LIN {X 0,Y 509.786,Z 447.475,A -85,B 0,C 180,E1 -5449.613,E2 -5449.613} C_VEL
LIN {X 0,Y 509.778,Z 447.48,A -85,B 0,C 180,E1 -5452.656,E2 -5452.656} C_VEL
LIN {X 0,Y 509.83,Z 447.482,A -85,B 0,C 180,E1 -5455.803,E2 -5455.803} C_VEL
LIN {X 0,Y 509.837,Z 447.476,A -85,B 0,C 180,E1 -5458.723,E2 -5458.723} C_VEL
LIN {X 0,Y 509.815,Z 447.48,A -85,B 0,C 180,E1 -5461.152,E2 -5461.152} C_VEL
LIN {X 0,Y 509.86,Z 447.686,A -85,B 0,C 180,E1 -5463.635,E2 -5463.635} C_VEL
LIN {X 0,Y 511.214,Z 455.666,A -85,B 0,C 180,E1 -5465.408,E2 -5465.408} C_VEL
LIN {X 0,Y 510.839,Z 468.185,A -85,B 0,C 180,E1 -5467.982,E2 -5467.982} C_VEL
LIN {X 0,Y 510.48,Z 482.835,A -85,B 0,C 180,E1 -5470.915,E2 -5470.915} C_VEL
LIN {X 0,Y 510.057,Z 498.364,A -85,B 0,C 180,E1 -5474.004,E2 -5474.004} C_VEL
LIN {X 0,Y 510.013,Z 500.382,A -85,B 0,C 180,E1 -5474.39,E2 -5474.39} C_VEL
LIN {X 0,Y 510.872,Z 505.663,A -85,B 0,C 180,E1 -5474.531,E2 -5474.531} C_VEL
LIN {X 0,Y 512.207,Z 513.365,A -85,B 0,C 180,E1 -5474.681,E2 -5474.681} C_VEL
LIN {X 0,Y 511.746,Z 605.354,A -85,B 0,C 180,E1 -5475.993,E2 -5475.993} C_VEL
LIN {X 0,Y 511.617,Z 615.274,A -85,B 0,C 180,E1 -5476.217,E2 -5476.217} C_VEL
LIN {X 0,Y 511.372,Z 625.264,A -85,B 0,C 180,E1 -5476.539,E2 -5476.539} C_VEL
LIN {X 0,Y 511.129,Z 635.625,A -85,B 0,C 180,E1 -5476.988,E2 -5476.988} C_VEL
LIN {X 0,Y 510.913,Z 644.923,A -85,B 0,C 180,E1 -5477.497,E2 -5477.497} C_VEL
LIN {X 0,Y 510.669,Z 653.783,A -85,B 0,C 180,E1 -5478.087,E2 -5478.087} C_VEL
LIN {X 0,Y 510.376,Z 662.514,A -85,B 0,C 180,E1 -5478.784,E2 -5478.784} C_VEL
LIN {X 0,Y 510.112,Z 669.938,A -85,B 0,C 180,E1 -5479.482,E2 -5479.482} C_VEL
LIN {X 0,Y 509.84,Z 678.737,A -85,B 0,C 180,E1 -5480.479,E2 -5480.479} C_VEL
LIN {X 0,Y 509.675,Z 684.729,A -85,B 0,C 180,E1 -5481.276,E2 -5481.276} C_VEL
LIN {X 0,Y 509.495,Z 691.04,A -85,B 0,C 180,E1 -5482.271,E2 -5482.271} C_VEL
LIN {X 0,Y 509.351,Z 697.115,A -85,B 0,C 180,E1 -5483.443,E2 -5483.443} C_VEL
LIN {X 0,Y 509.296,Z 701.404,A -85,B 0,C 180,E1 -5484.457,E2 -5484.457} C_VEL
LIN {X 0,Y 509.206,Z 705.362,A -85,B 0,C 180,E1 -5485.647,E2 -5485.647} C_VEL
LIN {X 0,Y 509.201,Z 708.291,A -85,B 0,C 180,E1 -5486.835,E2 -5486.835} C_VEL
LIN {X 0,Y 509.19,Z 709.788,A -85,B 0,C 180,E1 -5487.627,E2 -5487.627} C_VEL
LIN {X 0,Y 509.074,Z 711.303,A -85,B 0,C 180,E1 -5489.209,E2 -5489.209} C_VEL
LIN {X 0,Y 509.066,Z 711.581,A -85,B 0,C 180,E1 -5490,E2 -5490} C_VEL
LIN {X 0,Y 509.113,Z 710.71,A -85,B 0,C 180,E1 -5491.582,E2 -5491.582} C_VEL
LIN {X 0,Y 509.19,Z 709.788,A -85,B 0,C 180,E1 -5492.373,E2 -5492.373} C_VEL
LIN {X 0,Y 509.246,Z 706.45,A -85,B 0,C 180,E1 -5493.957,E2 -5493.957} C_VEL
LIN {X 0,Y 509.244,Z 702.829,A -85,B 0,C 180,E1 -5495.147,E2 -5495.147} C_VEL
LIN {X 0,Y 509.343,Z 699.891,A -85,B 0,C 180,E1 -5495.94,E2 -5495.94} C_VEL
LIN {X 0,Y 509.421,Z 694.317,A -85,B 0,C 180,E1 -5497.132,E2 -5497.132} C_VEL
LIN {X 0,Y 509.573,Z 688.665,A -85,B 0,C 180,E1 -5498.127,E2 -5498.127} C_VEL
LIN {X 0,Y 509.755,Z 681.86,A -85,B 0,C 180,E1 -5499.123,E2 -5499.123} C_VEL
LIN {X 0,Y 509.978,Z 673.64,A -85,B 0,C 180,E1 -5500.12,E2 -5500.12} C_VEL
LIN {X 0,Y 510.273,Z 665.811,A -85,B 0,C 180,E1 -5500.916,E2 -5500.916} C_VEL
LIN {X 0,Y 510.584,Z 657.725,A -85,B 0,C 180,E1 -5501.613,E2 -5501.613} C_VEL
LIN {X 0,Y 510.791,Z 647.557,A -85,B 0,C 180,E1 -5502.339,E2 -5502.339} C_VEL
LIN {X 0,Y 511.061,Z 639.564,A -85,B 0,C 180,E1 -5502.812,E2 -5502.812} C_VEL
LIN {X 0,Y 511.326,Z 629.054,A -85,B 0,C 180,E1 -5503.31,E2 -5503.31} C_VEL
LIN {X 0,Y 511.559,Z 618.719,A -85,B 0,C 180,E1 -5503.683,E2 -5503.683} C_VEL
LIN {X 0,Y 511.694,Z 607.997,A -85,B 0,C 180,E1 -5503.958,E2 -5503.958} C_VEL
LIN {X 0,Y 511.904,Z 585.223,A -85,B 0,C 180,E1 -5504.307,E2 -5504.307} C_VEL
LIN {X 0,Y 512.124,Z 512.714,A -85,B 0,C 180,E1 -5505.33,E2 -5505.33} C_VEL
LIN {X 0,Y 510.034,Z 500.586,A -85,B 0,C 180,E1 -5505.592,E2 -5505.592} C_VEL
LIN {X 0,Y 510.478,Z 483.881,A -85,B 0,C 180,E1 -5508.877,E2 -5508.877} C_VEL
LIN {X 0,Y 510.831,Z 469.232,A -85,B 0,C 180,E1 -5511.806,E2 -5511.806} C_VEL
LIN {X 0,Y 511.246,Z 456.791,A -85,B 0,C 180,E1 -5514.356,E2 -5514.356} C_VEL
LIN {X 0,Y 510.607,Z 451.626,A -85,B 0,C 180,E1 -5515.475,E2 -5515.475} C_VEL
LIN {X 0,Y 509.819,Z 447.591,A -85,B 0,C 180,E1 -5516.421,E2 -5516.421} C_VEL
LIN {X 0,Y 509.815,Z 447.48,A -85,B 0,C 180,E1 -5518.848,E2 -5518.848} C_VEL
LIN {X 0,Y 509.811,Z 447.481,A -85,B 0,C 180,E1 -5521.59,E2 -5521.59} C_VEL
LIN {X 0,Y 509.834,Z 447.478,A -85,B 0,C 180,E1 -5524.414,E2 -5524.414} C_VEL
LIN {X 0,Y 509.778,Z 447.48,A -85,B 0,C 180,E1 -5527.344,E2 -5527.344} C_VEL
LIN {X 0,Y 509.786,Z 447.475,A -85,B 0,C 180,E1 -5530.387,E2 -5530.387} C_VEL
LIN {X 0,Y 509.792,Z 447.48,A -85,B 0,C 180,E1 -5533.574,E2 -5533.574} C_VEL
LIN {X 0,Y 509.791,Z 447.483,A -85,B 0,C 180,E1 -5536.424,E2 -5536.424} C_VEL
LIN {X 0,Y 509.785,Z 447.481,A -85,B 0,C 180,E1 -5539.612,E2 -5539.612} C_VEL
LIN {X 0,Y 509.775,Z 447.482,A -85,B 0,C 180,E1 -5542.655,E2 -5542.655} C_VEL
LIN {X 0,Y 509.837,Z 447.474,A -85,B 0,C 180,E1 -5545.8,E2 -5545.8} C_VEL
LIN {X 0,Y 509.835,Z 447.474,A -85,B 0,C 180,E1 -5548.721,E2 -5548.721} C_VEL
LIN {X 0,Y 509.831,Z 447.472,A -85,B 0,C 180,E1 -5551.152,E2 -5551.152} C_VEL
LIN {X 0,Y 509.834,Z 447.469,A -85,B 0,C 180,E1 -5553.824,E2 -5553.824} C_VEL
LIN {X 0,Y 509.815,Z 447.479,A -85,B 0,C 180,E1 -5556.435,E2 -5556.435} C_VEL
LIN {X 0,Y 509.817,Z 447.475,A -85,B 0,C 180,E1 -5559.618,E2 -5559.618} C_VEL
LIN {X 0,Y 509.845,Z 447.471,A -85,B 0,C 180,E1 -5562.345,E2 -5562.345} C_VEL
LIN {X 0,Y 509.817,Z 447.477,A -85,B 0,C 180,E1 -5565.632,E2 -5565.632} C_VEL
LIN {X 0,Y 509.886,Z 447.469,A -85,B 0,C 180,E1 -5568.13,E2 -5568.13} C_VEL
LIN {X 0,Y 509.867,Z 447.458,A -85,B 0,C 180,E1 -5571.278,E2 -5571.278} C_VEL
LIN {X 0,Y 509.91,Z 447.463,A -85,B 0,C 180,E1 -5573.668,E2 -5573.668} C_VEL
LIN {X 0,Y 509.876,Z 447.467,A -85,B 0,C 180,E1 -5576.838,E2 -5576.838} C_VEL
LIN {X 0,Y 509.916,Z 447.46,A -85,B 0,C 180,E1 -5578.419,E2 -5578.419} C_VEL
LIN {X 0,Y 510.027,Z 447.445,A -85,B 0,C 180,E1 -5579.999,E2 -5579.999} C_VEL
LIN {X 0,Y 510.034,Z 447.45,A -85,B 0,C 180,E1 -5582.368,E2 -5582.368} C_VEL
LIN {X 0,Y 509.929,Z 447.463,A -85,B 0,C 180,E1 -5585.535,E2 -5585.535} C_VEL
LIN {X 0,Y 509.867,Z 447.474,A -85,B 0,C 180,E1 -5587.922,E2 -5587.922} C_VEL
LIN {X 0,Y 509.852,Z 447.463,A -85,B 0,C 180,E1 -5591.125,E2 -5591.125} C_VEL
LIN {X 0,Y 509.818,Z 447.475,A -85,B 0,C 180,E1 -5593.552,E2 -5593.552} C_VEL
LIN {X 0,Y 509.787,Z 447.487,A -85,B 0,C 180,E1 -5596.004,E2 -5596.004} C_VEL
LIN {X 0,Y 509.805,Z 447.469,A -85,B 0,C 180,E1 -5598.484,E2 -5598.484} C_VEL
LIN {X 0,Y 509.822,Z 447.471,A -85,B 0,C 180,E1 -5601.001,E2 -5601.001} C_VEL
LIN {X 0,Y 509.807,Z 447.479,A -85,B 0,C 180,E1 -5603.563,E2 -5603.563} C_VEL
LIN {X 0,Y 509.795,Z 447.475,A -85,B 0,C 180,E1 -5606.353,E2 -5606.353} C_VEL
LIN {X 0,Y 509.821,Z 447.472,A -85,B 0,C 180,E1 -5608.846,E2 -5608.846} C_VEL
LIN {X 0,Y 509.79,Z 447.482,A -85,B 0,C 180,E1 -5611.59,E2 -5611.59} C_VEL
LIN {X 0,Y 509.82,Z 447.473,A -85,B 0,C 180,E1 -5614.414,E2 -5614.414} C_VEL
LIN {X 0,Y 509.766,Z 447.483,A -85,B 0,C 180,E1 -5617.343,E2 -5617.343} C_VEL
LIN {X 0,Y 509.799,Z 447.477,A -85,B 0,C 180,E1 -5620.384,E2 -5620.384} C_VEL
LIN {X 0,Y 509.79,Z 447.481,A -85,B 0,C 180,E1 -5623.573,E2 -5623.573} C_VEL
LIN {X 0,Y 509.777,Z 447.473,A -85,B 0,C 180,E1 -5626.424,E2 -5626.424} C_VEL
LIN {X 0,Y 509.77,Z 447.475,A -85,B 0,C 180,E1 -5629.612,E2 -5629.612} C_VEL
LIN {X 0,Y 509.763,Z 447.483,A -85,B 0,C 180,E1 -5632.655,E2 -5632.655} C_VEL
LIN {X 0,Y 509.749,Z 447.486,A -85,B 0,C 180,E1 -5633.7,E2 -5633.7} C_VEL
LIN {X 0,Y 509.095,Z 447.56,A -85,B 0,C 180,E1 -5634.361,E2 -5634.361} C_VEL
LIN {X 0,Y 506.291,Z 447.907,A -85,B 0,C 180,E1 -5635.433,E2 -5635.433} C_VEL
LIN {X 0,Y 503.905,Z 448.213,A -85,B 0,C 180,E1 -5636.297,E2 -5636.297} C_VEL
LIN {X 0,Y 502.86,Z 448.341,A -85,B 0,C 180,E1 -5636.964,E2 -5636.964} C_VEL
LIN {X 0,Y 502.764,Z 448.353,A -85,B 0,C 180,E1 -5637.189,E2 -5637.189} C_VEL
LIN {X 0,Y 502.793,Z 448.35,A -85,B 0,C 180,E1 -5640.066,E2 -5640.066} C_VEL
LIN {X 0,Y 502.757,Z 448.358,A -85,B 0,C 180,E1 -5643.459,E2 -5643.459} C_VEL
LIN {X 0,Y 502.749,Z 448.364,A -85,B 0,C 180,E1 -5646.084,E2 -5646.084} C_VEL
LIN {X 0,Y 502.761,Z 448.357,A -85,B 0,C 180,E1 -5648.688,E2 -5648.688} C_VEL
LIN {X 0,Y 502.79,Z 448.353,A -85,B 0,C 180,E1 -5651.247,E2 -5651.247} C_VEL
LIN {X 0,Y 502.818,Z 448.35,A -85,B 0,C 180,E1 -5654.664,E2 -5654.664} C_VEL
LIN {X 0,Y 502.852,Z 448.351,A -85,B 0,C 180,E1 -5658.043,E2 -5658.043} C_VEL
LIN {X 0,Y 502.829,Z 448.349,A -85,B 0,C 180,E1 -5661.156,E2 -5661.156} C_VEL
LIN {X 0,Y 502.853,Z 448.349,A -85,B 0,C 180,E1 -5663.58,E2 -5663.58} C_VEL
LIN {X 0,Y 502.814,Z 448.351,A -85,B 0,C 180,E1 -5666.795,E2 -5666.795} C_VEL
LIN {X 0,Y 502.875,Z 448.346,A -85,B 0,C 180,E1 -5668.398,E2 -5668.398} C_VEL
LIN {X 0,Y 502.986,Z 448.335,A -85,B 0,C 180,E1 -5670,E2 -5670} C_VEL
LIN {X 0,Y 502.992,Z 448.331,A -85,B 0,C 180,E1 -5672.402,E2 -5672.402} C_VEL
LIN {X 0,Y 502.877,Z 448.346,A -85,B 0,C 180,E1 -5675.614,E2 -5675.614} C_VEL
LIN {X 0,Y 502.831,Z 448.354,A -85,B 0,C 180,E1 -5678.034,E2 -5678.034} C_VEL
LIN {X 0,Y 502.82,Z 448.35,A -85,B 0,C 180,E1 -5681.284,E2 -5681.284} C_VEL
LIN {X 0,Y 502.812,Z 448.352,A -85,B 0,C 180,E1 -5684.572,E2 -5684.572} C_VEL
LIN {X 0,Y 502.792,Z 448.359,A -85,B 0,C 180,E1 -5688.109,E2 -5688.109} C_VEL
LIN {X 0,Y 502.813,Z 448.351,A -85,B 0,C 180,E1 -5690.537,E2 -5690.537} C_VEL
LIN {X 0,Y 502.769,Z 448.355,A -85,B 0,C 180,E1 -5693.041,E2 -5693.041} C_VEL
LIN {X 0,Y 502.758,Z 448.361,A -85,B 0,C 180,E1 -5695.68,E2 -5695.68} C_VEL
LIN {X 0,Y 502.753,Z 448.353,A -85,B 0,C 180,E1 -5698.378,E2 -5698.378} C_VEL
LIN {X 0,Y 502.768,Z 448.354,A -85,B 0,C 180,E1 -5701.145,E2 -5701.145} C_VEL
LIN {X 0,Y 502.767,Z 448.35,A -85,B 0,C 180,E1 -5703.996,E2 -5703.996} C_VEL
LIN {X 0,Y 502.716,Z 448.36,A -85,B 0,C 180,E1 -5707.171,E2 -5707.171} C_VEL
LIN {X 0,Y 502.717,Z 448.358,A -85,B 0,C 180,E1 -5710.021,E2 -5710.021} C_VEL
LIN {X 0,Y 502.724,Z 448.348,A -85,B 0,C 180,E1 -5713.236,E2 -5713.236} C_VEL
LIN {X 0,Y 502.764,Z 448.356,A -85,B 0,C 180,E1 -5715.661,E2 -5715.661} C_VEL
LIN {X 0,Y 502.75,Z 448.351,A -85,B 0,C 180,E1 -5719.013,E2 -5719.013} C_VEL
LIN {X 0,Y 502.746,Z 448.364,A -85,B 0,C 180,E1 -5722.044,E2 -5722.044} C_VEL
LIN {X 0,Y 502.769,Z 448.348,A -85,B 0,C 180,E1 -5725.034,E2 -5725.034} C_VEL
LIN {X 0,Y 502.751,Z 448.362,A -85,B 0,C 180,E1 -5727.915,E2 -5727.915} C_VEL
LIN {X 0,Y 502.79,Z 448.348,A -85,B 0,C 180,E1 -5730.712,E2 -5730.712} C_VEL
LIN {X 0,Y 502.76,Z 448.349,A -85,B 0,C 180,E1 -5733.462,E2 -5733.462} C_VEL
LIN {X 0,Y 502.755,Z 448.362,A -85,B 0,C 180,E1 -5736.086,E2 -5736.086} C_VEL
LIN {X 0,Y 502.761,Z 448.351,A -85,B 0,C 180,E1 -5738.689,E2 -5738.689} C_VEL
LIN {X 0,Y 502.777,Z 448.35,A -85,B 0,C 180,E1 -5741.9,E2 -5741.9} C_VEL
LIN {X 0,Y 502.817,Z 448.349,A -85,B 0,C 180,E1 -5745.43,E2 -5745.43} C_VEL
LIN {X 0,Y 502.828,Z 448.337,A -85,B 0,C 180,E1 -5748.717,E2 -5748.717} C_VEL
LIN {X 0,Y 502.838,Z 448.346,A -85,B 0,C 180,E1 -5751.967,E2 -5751.967} C_VEL
LIN {X 0,Y 502.886,Z 448.341,A -85,B 0,C 180,E1 -5754.387,E2 -5754.387} C_VEL
LIN {X 0,Y 503.001,Z 448.325,A -85,B 0,C 180,E1 -5757.599,E2 -5757.599} C_VEL
LIN {X 0,Y 502.996,Z 448.32,A -85,B 0,C 180,E1 -5760.001,E2 -5760.001} C_VEL
LIN {X 0,Y 503.002,Z 448.325,A -85,B 0,C 180,E1 -5762.404,E2 -5762.404} C_VEL
LIN {X 0,Y 502.886,Z 448.343,A -85,B 0,C 180,E1 -5765.615,E2 -5765.615} C_VEL
LIN {X 0,Y 502.841,Z 448.34,A -85,B 0,C 180,E1 -5768.035,E2 -5768.035} C_VEL
LIN {X 0,Y 502.832,Z 448.34,A -85,B 0,C 180,E1 -5771.285,E2 -5771.285} C_VEL
LIN {X 0,Y 502.795,Z 448.349,A -85,B 0,C 180,E1 -5774.573,E2 -5774.573} C_VEL
LIN {X 0,Y 502.784,Z 448.346,A -85,B 0,C 180,E1 -5778.102,E2 -5778.102} C_VEL
LIN {X 0,Y 502.757,Z 448.353,A -85,B 0,C 180,E1 -5781.313,E2 -5781.313} C_VEL
LIN {X 0,Y 502.763,Z 448.359,A -85,B 0,C 180,E1 -5783.916,E2 -5783.916} C_VEL
LIN {X 0,Y 502.779,Z 448.344,A -85,B 0,C 180,E1 -5786.572,E2 -5786.572} C_VEL
LIN {X 0,Y 502.808,Z 448.357,A -85,B 0,C 180,E1 -5789.935,E2 -5789.935} C_VEL
LIN {X 0,Y 502.797,Z 448.346,A -85,B 0,C 180,E1 -5793.035,E2 -5793.035} C_VEL
LIN {X 0,Y 502.743,Z 448.363,A -85,B 0,C 180,E1 -5795.955,E2 -5795.955} C_VEL
LIN {X 0,Y 502.767,Z 448.351,A -85,B 0,C 180,E1 -5798.98,E2 -5798.98} C_VEL
LIN {X 0,Y 502.745,Z 448.361,A -85,B 0,C 180,E1 -5802.193,E2 -5802.193} C_VEL
LIN {X 0,Y 502.778,Z 448.355,A -85,B 0,C 180,E1 -5805.472,E2 -5805.472} C_VEL
LIN {X 0,Y 502.75,Z 448.347,A -85,B 0,C 180,E1 -5808.928,E2 -5808.928} C_VEL
LIN {X 0,Y 502.759,Z 448.36,A -85,B 0,C 180,E1 -5812.043,E2 -5812.043} C_VEL
LIN {X 0,Y 502.753,Z 448.355,A -85,B 0,C 180,E1 -5815.031,E2 -5815.031} C_VEL
LIN {X 0,Y 502.762,Z 448.36,A -85,B 0,C 180,E1 -5817.914,E2 -5817.914} C_VEL
LIN {X 0,Y 502.782,Z 448.356,A -85,B 0,C 180,E1 -5820.71,E2 -5820.71} C_VEL
LIN {X 0,Y 502.819,Z 448.562,A -85,B 0,C 180,E1 -5823.451,E2 -5823.451} C_VEL
LIN {X 0,Y 504.244,Z 456.649,A -85,B 0,C 180,E1 -5825.284,E2 -5825.284} C_VEL
LIN {X 0,Y 503.906,Z 468.046,A -85,B 0,C 180,E1 -5827.663,E2 -5827.663} C_VEL
LIN {X 0,Y 503.51,Z 481.652,A -85,B 0,C 180,E1 -5830.428,E2 -5830.428} C_VEL
LIN {X 0,Y 503.131,Z 495.1,A -85,B 0,C 180,E1 -5833.151,E2 -5833.151} C_VEL
LIN {X 0,Y 503.005,Z 500.389,A -85,B 0,C 180,E1 -5834.185,E2 -5834.185} C_VEL
LIN {X 0,Y 505.356,Z 514.508,A -85,B 0,C 180,E1 -5834.488,E2 -5834.488} C_VEL
LIN {X 0,Y 504.87,Z 605.158,A -85,B 0,C 180,E1 -5835.798,E2 -5835.798} C_VEL
LIN {X 0,Y 504.721,Z 615.078,A -85,B 0,C 180,E1 -5836.025,E2 -5836.025} C_VEL
LIN {X 0,Y 504.459,Z 625.067,A -85,B 0,C 180,E1 -5836.351,E2 -5836.351} C_VEL
LIN {X 0,Y 504.181,Z 635.428,A -85,B 0,C 180,E1 -5836.806,E2 -5836.806} C_VEL
LIN {X 0,Y 503.952,Z 645.118,A -85,B 0,C 180,E1 -5837.347,E2 -5837.347} C_VEL
LIN {X 0,Y 503.676,Z 653.586,A -85,B 0,C 180,E1 -5837.919,E2 -5837.919} C_VEL
LIN {X 0,Y 503.397,Z 662.317,A -85,B 0,C 180,E1 -5838.627,E2 -5838.627} C_VEL
LIN {X 0,Y 503.107,Z 669.741,A -85,B 0,C 180,E1 -5839.334,E2 -5839.334} C_VEL
LIN {X 0,Y 502.808,Z 678.54,A -85,B 0,C 180,E1 -5840.344,E2 -5840.344} C_VEL
LIN {X 0,Y 502.61,Z 684.531,A -85,B 0,C 180,E1 -5841.152,E2 -5841.152} C_VEL
LIN {X 0,Y 502.421,Z 690.843,A -85,B 0,C 180,E1 -5842.161,E2 -5842.161} C_VEL
LIN {X 0,Y 502.318,Z 696.295,A -85,B 0,C 180,E1 -5843.21,E2 -5843.21} C_VEL
LIN {X 0,Y 502.214,Z 701.207,A -85,B 0,C 180,E1 -5844.378,E2 -5844.378} C_VEL
LIN {X 0,Y 502.104,Z 705.165,A -85,B 0,C 180,E1 -5845.585,E2 -5845.585} C_VEL
LIN {X 0,Y 502.121,Z 708.095,A -85,B 0,C 180,E1 -5846.791,E2 -5846.791} C_VEL
LIN {X 0,Y 502.092,Z 709.591,A -85,B 0,C 180,E1 -5847.593,E2 -5847.593} C_VEL
LIN {X 0,Y 501.991,Z 711.107,A -85,B 0,C 180,E1 -5849.198,E2 -5849.198} C_VEL
LIN {X 0,Y 501.98,Z 711.385,A -85,B 0,C 180,E1 -5850,E2 -5850} C_VEL
LIN {X 0,Y 502.037,Z 710.515,A -85,B 0,C 180,E1 -5851.604,E2 -5851.604} C_VEL
LIN {X 0,Y 502.092,Z 709.591,A -85,B 0,C 180,E1 -5852.407,E2 -5852.407} C_VEL
LIN {X 0,Y 502.139,Z 706.253,A -85,B 0,C 180,E1 -5854.013,E2 -5854.013} C_VEL
LIN {X 0,Y 502.175,Z 702.633,A -85,B 0,C 180,E1 -5855.219,E2 -5855.219} C_VEL
LIN {X 0,Y 502.237,Z 697.904,A -85,B 0,C 180,E1 -5856.427,E2 -5856.427} C_VEL
LIN {X 0,Y 502.362,Z 693.027,A -85,B 0,C 180,E1 -5857.435,E2 -5857.435} C_VEL
LIN {X 0,Y 502.529,Z 687.155,A -85,B 0,C 180,E1 -5858.444,E2 -5858.444} C_VEL
LIN {X 0,Y 502.699,Z 681.662,A -85,B 0,C 180,E1 -5859.252,E2 -5859.252} C_VEL
LIN {X 0,Y 502.958,Z 673.443,A -85,B 0,C 180,E1 -5860.262,E2 -5860.262} C_VEL
LIN {X 0,Y 503.276,Z 665.614,A -85,B 0,C 180,E1 -5861.07,E2 -5861.07} C_VEL
LIN {X 0,Y 503.605,Z 657.528,A -85,B 0,C 180,E1 -5861.777,E2 -5861.777} C_VEL
LIN {X 0,Y 503.803,Z 648.403,A -85,B 0,C 180,E1 -5862.446,E2 -5862.446} C_VEL
LIN {X 0,Y 504.119,Z 639.367,A -85,B 0,C 180,E1 -5862.991,E2 -5862.991} C_VEL
LIN {X 0,Y 504.42,Z 628.858,A -85,B 0,C 180,E1 -5863.496,E2 -5863.496} C_VEL
LIN {X 0,Y 504.664,Z 618.523,A -85,B 0,C 180,E1 -5863.874,E2 -5863.874} C_VEL
LIN {X 0,Y 504.803,Z 607.8,A -85,B 0,C 180,E1 -5864.153,E2 -5864.153} C_VEL
LIN {X 0,Y 505.041,Z 585.027,A -85,B 0,C 180,E1 -5864.506,E2 -5864.506} C_VEL
LIN {X 0,Y 505.312,Z 513.673,A -85,B 0,C 180,E1 -5865.526,E2 -5865.526} C_VEL
LIN {X 0,Y 503.03,Z 500.529,A -85,B 0,C 180,E1 -5865.806,E2 -5865.806} C_VEL
LIN {X 0,Y 503.006,Z 499.492,A -85,B 0,C 180,E1 -5865.945,E2 -5865.945} C_VEL
LIN {X 0,Y 503.457,Z 484.79,A -85,B 0,C 180,E1 -5868.939,E2 -5868.939} C_VEL
LIN {X 0,Y 503.874,Z 469.094,A -85,B 0,C 180,E1 -5872.123,E2 -5872.123} C_VEL
LIN {X 0,Y 504.288,Z 457.707,A -85,B 0,C 180,E1 -5874.494,E2 -5874.494} C_VEL
LIN {X 0,Y 503.382,Z 451.532,A -85,B 0,C 180,E1 -5875.863,E2 -5875.863} C_VEL
LIN {X 0,Y 502.788,Z 448.45,A -85,B 0,C 180,E1 -5876.626,E2 -5876.626} C_VEL
LIN {X 0,Y 502.79,Z 448.356,A -85,B 0,C 180,E1 -5879.929,E2 -5879.929} C_VEL
LIN {X 0,Y 502.804,Z 448.348,A -85,B 0,C 180,E1 -5883.033,E2 -5883.033} C_VEL
LIN {X 0,Y 502.744,Z 448.358,A -85,B 0,C 180,E1 -5885.953,E2 -5885.953} C_VEL
LIN {X 0,Y 502.774,Z 448.353,A -85,B 0,C 180,E1 -5888.978,E2 -5888.978} C_VEL
LIN {X 0,Y 502.745,Z 448.359,A -85,B 0,C 180,E1 -5892.191,E2 -5892.191} C_VEL
LIN {X 0,Y 502.778,Z 448.352,A -85,B 0,C 180,E1 -5895.47,E2 -5895.47} C_VEL
LIN {X 0,Y 502.749,Z 448.355,A -85,B 0,C 180,E1 -5898.926,E2 -5898.926} C_VEL
LIN {X 0,Y 502.754,Z 448.361,A -85,B 0,C 180,E1 -5902.042,E2 -5902.042} C_VEL
LIN {X 0,Y 502.781,Z 448.348,A -85,B 0,C 180,E1 -5905.032,E2 -5905.032} C_VEL
LIN {X 0,Y 502.762,Z 448.356,A -85,B 0,C 180,E1 -5907.913,E2 -5907.913} C_VEL
LIN {X 0,Y 502.801,Z 448.349,A -85,B 0,C 180,E1 -5910.71,E2 -5910.71} C_VEL
LIN {X 0,Y 502.77,Z 448.345,A -85,B 0,C 180,E1 -5913.459,E2 -5913.459} C_VEL
LIN {X 0,Y 502.763,Z 448.359,A -85,B 0,C 180,E1 -5916.084,E2 -5916.084} C_VEL
LIN {X 0,Y 502.757,Z 448.353,A -85,B 0,C 180,E1 -5918.687,E2 -5918.687} C_VEL
LIN {X 0,Y 502.784,Z 448.346,A -85,B 0,C 180,E1 -5921.898,E2 -5921.898} C_VEL
LIN {X 0,Y 502.795,Z 448.349,A -85,B 0,C 180,E1 -5925.427,E2 -5925.427} C_VEL
LIN {X 0,Y 502.832,Z 448.34,A -85,B 0,C 180,E1 -5928.715,E2 -5928.715} C_VEL
LIN {X 0,Y 502.841,Z 448.34,A -85,B 0,C 180,E1 -5931.965,E2 -5931.965} C_VEL
LIN {X 0,Y 502.886,Z 448.343,A -85,B 0,C 180,E1 -5934.385,E2 -5934.385} C_VEL
LIN {X 0,Y 503.002,Z 448.325,A -85,B 0,C 180,E1 -5937.596,E2 -5937.596} C_VEL
LIN {X 0,Y 502.996,Z 448.32,A -85,B 0,C 180,E1 -5939.999,E2 -5939.999} C_VEL
LIN {X 0,Y 503.001,Z 448.325,A -85,B 0,C 180,E1 -5942.401,E2 -5942.401} C_VEL
LIN {X 0,Y 502.886,Z 448.341,A -85,B 0,C 180,E1 -5945.613,E2 -5945.613} C_VEL
LIN {X 0,Y 502.838,Z 448.346,A -85,B 0,C 180,E1 -5948.033,E2 -5948.033} C_VEL
LIN {X 0,Y 502.828,Z 448.337,A -85,B 0,C 180,E1 -5951.283,E2 -5951.283} C_VEL
LIN {X 0,Y 502.817,Z 448.349,A -85,B 0,C 180,E1 -5954.57,E2 -5954.57} C_VEL
LIN {X 0,Y 502.777,Z 448.35,A -85,B 0,C 180,E1 -5958.1,E2 -5958.1} C_VEL
LIN {X 0,Y 502.761,Z 448.351,A -85,B 0,C 180,E1 -5961.311,E2 -5961.311} C_VEL
LIN {X 0,Y 502.755,Z 448.362,A -85,B 0,C 180,E1 -5963.914,E2 -5963.914} C_VEL
LIN {X 0,Y 502.77,Z 448.347,A -85,B 0,C 180,E1 -5966.57,E2 -5966.57} C_VEL
LIN {X 0,Y 502.797,Z 448.354,A -85,B 0,C 180,E1 -5969.933,E2 -5969.933} C_VEL
LIN {X 0,Y 502.786,Z 448.349,A -85,B 0,C 180,E1 -5973.033,E2 -5973.033} C_VEL
LIN {X 0,Y 502.731,Z 448.36,A -85,B 0,C 180,E1 -5975.953,E2 -5975.953} C_VEL
LIN {X 0,Y 502.769,Z 448.353,A -85,B 0,C 180,E1 -5978.977,E2 -5978.977} C_VEL
LIN {X 0,Y 502.73,Z 448.365,A -85,B 0,C 180,E1 -5982.191,E2 -5982.191} C_VEL
LIN {X 0,Y 502.763,Z 448.354,A -85,B 0,C 180,E1 -5985.47,E2 -5985.47} C_VEL
LIN {X 0,Y 502.734,Z 448.348,A -85,B 0,C 180,E1 -5988.926,E2 -5988.926} C_VEL
LIN {X 0,Y 502.743,Z 448.366,A -85,B 0,C 180,E1 -5992.042,E2 -5992.042} C_VEL
LIN {X 0,Y 502.766,Z 448.344,A -85,B 0,C 180,E1 -5995.032,E2 -5995.032} C_VEL
LIN {X 0,Y 502.764,Z 448.353,A -85,B 0,C 180,E1 -5997.189,E2 -5997.189} C_VEL
LIN {X 0,Y 502.071,Z 448.447,A -85,B 0,C 180,E1 -5997.858,E2 -5997.858} C_VEL
LIN {X 0,Y 499.221,Z 448.795,A -85,B 0,C 180,E1 -5998.944,E2 -5998.944} C_VEL
LIN {X 0,Y 496.826,Z 449.096,A -85,B 0,C 180,E1 -5999.82,E2 -5999.82} C_VEL
LIN {X 0,Y 495.794,Z 449.218,A -85,B 0,C 180,E1 -6000.495,E2 -6000.495} C_VEL
LIN {X 0,Y 495.707,Z 449.227,A -85,B 0,C 180,E1 -6000.724,E2 -6000.724} C_VEL
LIN {X 0,Y 495.699,Z 449.242,A -85,B 0,C 180,E1 -6003.927,E2 -6003.927} C_VEL
LIN {X 0,Y 495.741,Z 449.231,A -85,B 0,C 180,E1 -6007.14,E2 -6007.14} C_VEL
LIN {X 0,Y 495.743,Z 449.237,A -85,B 0,C 180,E1 -6010.109,E2 -6010.109} C_VEL
LIN {X 0,Y 495.692,Z 449.239,A -85,B 0,C 180,E1 -6012.678,E2 -6012.678} C_VEL
LIN {X 0,Y 495.762,Z 449.229,A -85,B 0,C 180,E1 -6015.216,E2 -6015.216} C_VEL
LIN {X 0,Y 495.804,Z 449.226,A -85,B 0,C 180,E1 -6018.554,E2 -6018.554} C_VEL
LIN {X 0,Y 495.795,Z 449.23,A -85,B 0,C 180,E1 -6021.851,E2 -6021.851} C_VEL
LIN {X 0,Y 495.836,Z 449.224,A -85,B 0,C 180,E1 -6024.306,E2 -6024.306} C_VEL
LIN {X 0,Y 495.959,Z 449.207,A -85,B 0,C 180,E1 -6027.564,E2 -6027.564} C_VEL
LIN {X 0,Y 495.955,Z 449.211,A -85,B 0,C 180,E1 -6030,E2 -6030} C_VEL
LIN {X 0,Y 495.959,Z 449.207,A -85,B 0,C 180,E1 -6032.436,E2 -6032.436} C_VEL
LIN {X 0,Y 495.836,Z 449.224,A -85,B 0,C 180,E1 -6035.694,E2 -6035.694} C_VEL
LIN {X 0,Y 495.795,Z 449.23,A -85,B 0,C 180,E1 -6038.149,E2 -6038.149} C_VEL
LIN {X 0,Y 495.804,Z 449.226,A -85,B 0,C 180,E1 -6041.446,E2 -6041.446} C_VEL
LIN {X 0,Y 495.762,Z 449.229,A -85,B 0,C 180,E1 -6044.784,E2 -6044.784} C_VEL
LIN {X 0,Y 495.755,Z 449.234,A -85,B 0,C 180,E1 -6048.235,E2 -6048.235} C_VEL
LIN {X 0,Y 495.758,Z 449.229,A -85,B 0,C 180,E1 -6050.757,E2 -6050.757} C_VEL
LIN {X 0,Y 495.721,Z 449.234,A -85,B 0,C 180,E1 -6053.388,E2 -6053.388} C_VEL
LIN {X 0,Y 495.721,Z 449.233,A -85,B 0,C 180,E1 -6056.73,E2 -6056.73} C_VEL
LIN {X 0,Y 495.739,Z 449.226,A -85,B 0,C 180,E1 -6059.748,E2 -6059.748} C_VEL
LIN {X 0,Y 495.726,Z 449.231,A -85,B 0,C 180,E1 -6062.597,E2 -6062.597} C_VEL
LIN {X 0,Y 495.712,Z 449.225,A -85,B 0,C 180,E1 -6065.54,E2 -6065.54} C_VEL
LIN {X 0,Y 495.718,Z 449.232,A -85,B 0,C 180,E1 -6068.765,E2 -6068.765} C_VEL
LIN {X 0,Y 495.686,Z 449.224,A -85,B 0,C 180,E1 -6071.788,E2 -6071.788} C_VEL
LIN {X 0,Y 495.721,Z 449.229,A -85,B 0,C 180,E1 -6075.142,E2 -6075.142} C_VEL
LIN {X 0,Y 495.709,Z 449.233,A -85,B 0,C 180,E1 -6078.216,E2 -6078.216} C_VEL
LIN {X 0,Y 495.726,Z 449.231,A -85,B 0,C 180,E1 -6081.236,E2 -6081.236} C_VEL
LIN {X 0,Y 495.715,Z 449.228,A -85,B 0,C 180,E1 -6084.462,E2 -6084.462} C_VEL
LIN {X 0,Y 495.73,Z 449.23,A -85,B 0,C 180,E1 -6087.405,E2 -6087.405} C_VEL
LIN {X 0,Y 495.744,Z 449.23,A -85,B 0,C 180,E1 -6090.254,E2 -6090.254} C_VEL
LIN {X 0,Y 495.726,Z 449.223,A -85,B 0,C 180,E1 -6093.272,E2 -6093.272} C_VEL
LIN {X 0,Y 495.728,Z 449.231,A -85,B 0,C 180,E1 -6096.613,E2 -6096.613} C_VEL
LIN {X 0,Y 495.758,Z 449.224,A -85,B 0,C 180,E1 -6099.329,E2 -6099.329} C_VEL
LIN {X 0,Y 495.726,Z 449.226,A -85,B 0,C 180,E1 -6101.828,E2 -6101.828} C_VEL
LIN {X 0,Y 495.767,Z 449.226,A -85,B 0,C 180,E1 -6105.218,E2 -6105.218} C_VEL
LIN {X 0,Y 495.813,Z 449.212,A -85,B 0,C 180,E1 -6108.555,E2 -6108.555} C_VEL
LIN {X 0,Y 495.802,Z 449.22,A -85,B 0,C 180,E1 -6111.852,E2 -6111.852} C_VEL
LIN {X 0,Y 495.844,Z 449.219,A -85,B 0,C 180,E1 -6114.307,E2 -6114.307} C_VEL
LIN {X 0,Y 495.968,Z 449.201,A -85,B 0,C 180,E1 -6117.565,E2 -6117.565} C_VEL
LIN {X 0,Y 495.965,Z 449.195,A -85,B 0,C 180,E1 -6120.001,E2 -6120.001} C_VEL
LIN {X 0,Y 495.969,Z 449.201,A -85,B 0,C 180,E1 -6122.438,E2 -6122.438} C_VEL
LIN {X 0,Y 495.844,Z 449.221,A -85,B 0,C 180,E1 -6125.695,E2 -6125.695} C_VEL
LIN {X 0,Y 495.805,Z 449.214,A -85,B 0,C 180,E1 -6128.15,E2 -6128.15} C_VEL
LIN {X 0,Y 495.817,Z 449.215,A -85,B 0,C 180,E1 -6131.447,E2 -6131.447} C_VEL
LIN {X 0,Y 495.743,Z 449.227,A -85,B 0,C 180,E1 -6134.785,E2 -6134.785} C_VEL
LIN {X 0,Y 495.745,Z 449.221,A -85,B 0,C 180,E1 -6138.227,E2 -6138.227} C_VEL
LIN {X 0,Y 495.724,Z 449.233,A -85,B 0,C 180,E1 -6141.631,E2 -6141.631} C_VEL
LIN {X 0,Y 495.709,Z 449.232,A -85,B 0,C 180,E1 -6144.278,E2 -6144.278} C_VEL
LIN {X 0,Y 495.726,Z 449.221,A -85,B 0,C 180,E1 -6146.98,E2 -6146.98} C_VEL
LIN {X 0,Y 495.755,Z 449.232,A -85,B 0,C 180,E1 -6150.146,E2 -6150.146} C_VEL
LIN {X 0,Y 495.747,Z 449.224,A -85,B 0,C 180,E1 -6153.237,E2 -6153.237} C_VEL
LIN {X 0,Y 495.685,Z 449.242,A -85,B 0,C 180,E1 -6156.084,E2 -6156.084} C_VEL
LIN {X 0,Y 495.728,Z 449.228,A -85,B 0,C 180,E1 -6158.764,E2 -6158.764} C_VEL
LIN {X 0,Y 495.699,Z 449.24,A -85,B 0,C 180,E1 -6161.788,E2 -6161.788} C_VEL
LIN {X 0,Y 495.731,Z 449.23,A -85,B 0,C 180,E1 -6165.143,E2 -6165.143} C_VEL
LIN {X 0,Y 495.702,Z 449.229,A -85,B 0,C 180,E1 -6168.214,E2 -6168.214} C_VEL
LIN {X 0,Y 495.719,Z 449.234,A -85,B 0,C 180,E1 -6171.406,E2 -6171.406} C_VEL
LIN {X 0,Y 495.716,Z 449.234,A -85,B 0,C 180,E1 -6174.46,E2 -6174.46} C_VEL
LIN {X 0,Y 495.728,Z 449.231,A -85,B 0,C 180,E1 -6177.403,E2 -6177.403} C_VEL
LIN {X 0,Y 495.737,Z 449.236,A -85,B 0,C 180,E1 -6180.252,E2 -6180.252} C_VEL
LIN {X 0,Y 495.777,Z 449.445,A -85,B 0,C 180,E1 -6183.263,E2 -6183.263} C_VEL
LIN {X 0,Y 497.32,Z 458.587,A -85,B 0,C 180,E1 -6185.362,E2 -6185.362} C_VEL
LIN {X 0,Y 496.84,Z 473.145,A -85,B 0,C 180,E1 -6188.421,E2 -6188.421} C_VEL
LIN {X 0,Y 496.305,Z 489.769,A -85,B 0,C 180,E1 -6191.849,E2 -6191.849} C_VEL
LIN {X 0,Y 495.996,Z 500.008,A -85,B 0,C 180,E1 -6193.94,E2 -6193.94} C_VEL
LIN {X 0,Y 496.935,Z 505.811,A -85,B 0,C 180,E1 -6194.094,E2 -6194.094} C_VEL
LIN {X 0,Y 498.517,Z 515.722,A -85,B 0,C 180,E1 -6194.29,E2 -6194.29} C_VEL
LIN {X 0,Y 498.001,Z 604.962,A -85,B 0,C 180,E1 -6195.598,E2 -6195.598} C_VEL
LIN {X 0,Y 497.836,Z 614.882,A -85,B 0,C 180,E1 -6195.828,E2 -6195.828} C_VEL
LIN {X 0,Y 497.562,Z 624.871,A -85,B 0,C 180,E1 -6196.158,E2 -6196.158} C_VEL
LIN {X 0,Y 497.263,Z 635.231,A -85,B 0,C 180,E1 -6196.619,E2 -6196.619} C_VEL
LIN {X 0,Y 497.015,Z 643.945,A -85,B 0,C 180,E1 -6197.103,E2 -6197.103} C_VEL
LIN {X 0,Y 496.711,Z 653.389,A -85,B 0,C 180,E1 -6197.747,E2 -6197.747} C_VEL
LIN {X 0,Y 496.429,Z 662.121,A -85,B 0,C 180,E1 -6198.465,E2 -6198.465} C_VEL
LIN {X 0,Y 496.111,Z 669.544,A -85,B 0,C 180,E1 -6199.181,E2 -6199.181} C_VEL
LIN {X 0,Y 495.759,Z 678.342,A -85,B 0,C 180,E1 -6200.206,E2 -6200.206} C_VEL
LIN {X 0,Y 495.572,Z 684.335,A -85,B 0,C 180,E1 -6201.025,E2 -6201.025} C_VEL
LIN {X 0,Y 495.371,Z 690.646,A -85,B 0,C 180,E1 -6202.049,E2 -6202.049} C_VEL
LIN {X 0,Y 495.253,Z 695.919,A -85,B 0,C 180,E1 -6203.072,E2 -6203.072} C_VEL
LIN {X 0,Y 495.131,Z 701.01,A -85,B 0,C 180,E1 -6204.298,E2 -6204.298} C_VEL
LIN {X 0,Y 495.01,Z 704.968,A -85,B 0,C 180,E1 -6205.521,E2 -6205.521} C_VEL
LIN {X 0,Y 495.042,Z 707.899,A -85,B 0,C 180,E1 -6206.745,E2 -6206.745} C_VEL
LIN {X 0,Y 494.999,Z 709.395,A -85,B 0,C 180,E1 -6207.559,E2 -6207.559} C_VEL
LIN {X 0,Y 494.911,Z 710.911,A -85,B 0,C 180,E1 -6209.186,E2 -6209.186} C_VEL
LIN {X 0,Y 494.898,Z 711.189,A -85,B 0,C 180,E1 -6210,E2 -6210} C_VEL
LIN {X 0,Y 494.963,Z 710.319,A -85,B 0,C 180,E1 -6211.627,E2 -6211.627} C_VEL
LIN {X 0,Y 494.999,Z 709.395,A -85,B 0,C 180,E1 -6212.441,E2 -6212.441} C_VEL
LIN {X 0,Y 495.033,Z 706.056,A -85,B 0,C 180,E1 -6214.071,E2 -6214.071} C_VEL
LIN {X 0,Y 495.108,Z 702.436,A -85,B 0,C 180,E1 -6215.294,E2 -6215.294} C_VEL
LIN {X 0,Y 495.137,Z 698.885,A -85,B 0,C 180,E1 -6216.251,E2 -6216.251} C_VEL
LIN {X 0,Y 495.31,Z 692.831,A -85,B 0,C 180,E1 -6217.542,E2 -6217.542} C_VEL
LIN {X 0,Y 495.484,Z 686.958,A -85,B 0,C 180,E1 -6218.565,E2 -6218.565} C_VEL
LIN {X 0,Y 495.645,Z 681.465,A -85,B 0,C 180,E1 -6219.385,E2 -6219.385} C_VEL
LIN {X 0,Y 495.944,Z 673.245,A -85,B 0,C 180,E1 -6220.409,E2 -6220.409} C_VEL
LIN {X 0,Y 496.274,Z 665.417,A -85,B 0,C 180,E1 -6221.228,E2 -6221.228} C_VEL
LIN {X 0,Y 496.63,Z 657.331,A -85,B 0,C 180,E1 -6221.944,E2 -6221.944} C_VEL
LIN {X 0,Y 496.848,Z 648.479,A -85,B 0,C 180,E1 -6222.605,E2 -6222.605} C_VEL
LIN {X 0,Y 497.174,Z 639.17,A -85,B 0,C 180,E1 -6223.176,E2 -6223.176} C_VEL
LIN {X 0,Y 497.517,Z 628.661,A -85,B 0,C 180,E1 -6223.687,E2 -6223.687} C_VEL
LIN {X 0,Y 497.788,Z 618.327,A -85,B 0,C 180,E1 -6224.07,E2 -6224.07} C_VEL
LIN {X 0,Y 497.908,Z 607.604,A -85,B 0,C 180,E1 -6224.353,E2 -6224.353} C_VEL
LIN {X 0,Y 498.16,Z 588.411,A -85,B 0,C 180,E1 -6224.659,E2 -6224.659} C_VEL
LIN {X 0,Y 498.352,Z 514.018,A -85,B 0,C 180,E1 -6225.74,E2 -6225.74} C_VEL
LIN {X 0,Y 496.007,Z 500.256,A -85,B 0,C 180,E1 -6226.04,E2 -6226.04} C_VEL
LIN {X 0,Y 496.002,Z 497.989,A -85,B 0,C 180,E1 -6226.462,E2 -6226.462} C_VEL
LIN {X 0,Y 496.465,Z 484.653,A -85,B 0,C 180,E1 -6229.216,E2 -6229.216} C_VEL
LIN {X 0,Y 496.953,Z 468.955,A -85,B 0,C 180,E1 -6232.447,E2 -6232.447} C_VEL
LIN {X 0,Y 497.324,Z 458.627,A -85,B 0,C 180,E1 -6234.638,E2 -6234.638} C_VEL
LIN {X 0,Y 496.054,Z 450.903,A -85,B 0,C 180,E1 -6236.386,E2 -6236.386} C_VEL
LIN {X 0,Y 495.764,Z 449.326,A -85,B 0,C 180,E1 -6236.812,E2 -6236.812} C_VEL
LIN {X 0,Y 495.742,Z 449.233,A -85,B 0,C 180,E1 -6240.141,E2 -6240.141} C_VEL
LIN {X 0,Y 495.753,Z 449.226,A -85,B 0,C 180,E1 -6243.236,E2 -6243.236} C_VEL
LIN {X 0,Y 495.687,Z 449.237,A -85,B 0,C 180,E1 -6246.082,E2 -6246.082} C_VEL
LIN {X 0,Y 495.734,Z 449.231,A -85,B 0,C 180,E1 -6248.763,E2 -6248.763} C_VEL
LIN {X 0,Y 495.702,Z 449.229,A -85,B 0,C 180,E1 -6251.786,E2 -6251.786} C_VEL
LIN {X 0,Y 495.731,Z 449.229,A -85,B 0,C 180,E1 -6255.141,E2 -6255.141} C_VEL
LIN {X 0,Y 495.699,Z 449.24,A -85,B 0,C 180,E1 -6258.212,E2 -6258.212} C_VEL
LIN {X 0,Y 495.713,Z 449.231,A -85,B 0,C 180,E1 -6261.404,E2 -6261.404} C_VEL
LIN {X 0,Y 495.727,Z 449.23,A -85,B 0,C 180,E1 -6264.46,E2 -6264.46} C_VEL
LIN {X 0,Y 495.741,Z 449.225,A -85,B 0,C 180,E1 -6267.403,E2 -6267.403} C_VEL
LIN {X 0,Y 495.755,Z 449.232,A -85,B 0,C 180,E1 -6270.252,E2 -6270.252} C_VEL
LIN {X 0,Y 495.735,Z 449.22,A -85,B 0,C 180,E1 -6273.27,E2 -6273.27} C_VEL
LIN {X 0,Y 495.736,Z 449.231,A -85,B 0,C 180,E1 -6276.611,E2 -6276.611} C_VEL
LIN {X 0,Y 495.722,Z 449.229,A -85,B 0,C 180,E1 -6279.34,E2 -6279.34} C_VEL
LIN {X 0,Y 495.731,Z 449.223,A -85,B 0,C 180,E1 -6281.825,E2 -6281.825} C_VEL
LIN {X 0,Y 495.743,Z 449.227,A -85,B 0,C 180,E1 -6285.215,E2 -6285.215} C_VEL
LIN {X 0,Y 495.817,Z 449.215,A -85,B 0,C 180,E1 -6288.553,E2 -6288.553} C_VEL
LIN {X 0,Y 495.805,Z 449.214,A -85,B 0,C 180,E1 -6291.85,E2 -6291.85} C_VEL
LIN {X 0,Y 495.844,Z 449.221,A -85,B 0,C 180,E1 -6294.305,E2 -6294.305} C_VEL
LIN {X 0,Y 495.969,Z 449.201,A -85,B 0,C 180,E1 -6297.562,E2 -6297.562} C_VEL
LIN {X 0,Y 495.965,Z 449.195,A -85,B 0,C 180,E1 -6299.999,E2 -6299.999} C_VEL
LIN {X 0,Y 495.968,Z 449.201,A -85,B 0,C 180,E1 -6302.435,E2 -6302.435} C_VEL
LIN {X 0,Y 495.844,Z 449.219,A -85,B 0,C 180,E1 -6305.693,E2 -6305.693} C_VEL
LIN {X 0,Y 495.802,Z 449.22,A -85,B 0,C 180,E1 -6308.148,E2 -6308.148} C_VEL
LIN {X 0,Y 495.813,Z 449.212,A -85,B 0,C 180,E1 -6311.445,E2 -6311.445} C_VEL
LIN {X 0,Y 495.767,Z 449.226,A -85,B 0,C 180,E1 -6314.782,E2 -6314.782} C_VEL
LIN {X 0,Y 495.738,Z 449.224,A -85,B 0,C 180,E1 -6318.225,E2 -6318.225} C_VEL
LIN {X 0,Y 495.755,Z 449.223,A -85,B 0,C 180,E1 -6320.756,E2 -6320.756} C_VEL
LIN {X 0,Y 495.728,Z 449.231,A -85,B 0,C 180,E1 -6323.387,E2 -6323.387} C_VEL
LIN {X 0,Y 495.726,Z 449.223,A -85,B 0,C 180,E1 -6326.728,E2 -6326.728} C_VEL
LIN {X 0,Y 495.744,Z 449.23,A -85,B 0,C 180,E1 -6329.746,E2 -6329.746} C_VEL
LIN {X 0,Y 495.73,Z 449.23,A -85,B 0,C 180,E1 -6332.595,E2 -6332.595} C_VEL
LIN {X 0,Y 495.715,Z 449.228,A -85,B 0,C 180,E1 -6335.538,E2 -6335.538} C_VEL
LIN {X 0,Y 495.726,Z 449.231,A -85,B 0,C 180,E1 -6338.764,E2 -6338.764} C_VEL
LIN {X 0,Y 495.709,Z 449.233,A -85,B 0,C 180,E1 -6341.784,E2 -6341.784} C_VEL
LIN {X 0,Y 495.718,Z 449.229,A -85,B 0,C 180,E1 -6345.141,E2 -6345.141} C_VEL
LIN {X 0,Y 495.686,Z 449.224,A -85,B 0,C 180,E1 -6348.212,E2 -6348.212} C_VEL
LIN {X 0,Y 495.703,Z 449.234,A -85,B 0,C 180,E1 -6351.404,E2 -6351.404} C_VEL
LIN {X 0,Y 495.712,Z 449.225,A -85,B 0,C 180,E1 -6354.46,E2 -6354.46} C_VEL
LIN {X 0,Y 495.726,Z 449.231,A -85,B 0,C 180,E1 -6357.403,E2 -6357.403} C_VEL
LIN {X 0,Y 495.739,Z 449.226,A -85,B 0,C 180,E1 -6360.252,E2 -6360.252} C_VEL
LIN {X 0,Y 495.707,Z 449.227,A -85,B 0,C 180,E1 -6360.724,E2 -6360.724} C_VEL
LIN {X 0,Y 495.026,Z 449.314,A -85,B 0,C 180,E1 -6361.403,E2 -6361.403} C_VEL
LIN {X 0,Y 492.15,Z 449.68,A -85,B 0,C 180,E1 -6362.505,E2 -6362.505} C_VEL
LIN {X 0,Y 489.742,Z 449.979,A -85,B 0,C 180,E1 -6363.393,E2 -6363.393} C_VEL
LIN {X 0,Y 488.733,Z 450.11,A -85,B 0,C 180,E1 -6364.079,E2 -6364.079} C_VEL
LIN {X 0,Y 488.664,Z 450.114,A -85,B 0,C 180,E1 -6364.311,E2 -6364.311} C_VEL
LIN {X 0,Y 488.704,Z 450.107,A -85,B 0,C 180,E1 -6367.152,E2 -6367.152} C_VEL
LIN {X 0,Y 488.702,Z 450.113,A -85,B 0,C 180,E1 -6369.81,E2 -6369.81} C_VEL
LIN {X 0,Y 488.661,Z 450.117,A -85,B 0,C 180,E1 -6372.421,E2 -6372.421} C_VEL
LIN {X 0,Y 488.731,Z 450.105,A -85,B 0,C 180,E1 -6374.999,E2 -6374.999} C_VEL
LIN {X 0,Y 488.767,Z 450.104,A -85,B 0,C 180,E1 -6378.387,E2 -6378.387} C_VEL
LIN {X 0,Y 488.743,Z 450.108,A -85,B 0,C 180,E1 -6381.732,E2 -6381.732} C_VEL
LIN {X 0,Y 488.795,Z 450.102,A -85,B 0,C 180,E1 -6384.224,E2 -6384.224} C_VEL
LIN {X 0,Y 488.925,Z 450.084,A -85,B 0,C 180,E1 -6387.528,E2 -6387.528} C_VEL
LIN {X 0,Y 488.924,Z 450.086,A -85,B 0,C 180,E1 -6390,E2 -6390} C_VEL
LIN {X 0,Y 488.925,Z 450.083,A -85,B 0,C 180,E1 -6392.472,E2 -6392.472} C_VEL
LIN {X 0,Y 488.795,Z 450.102,A -85,B 0,C 180,E1 -6395.776,E2 -6395.776} C_VEL
LIN {X 0,Y 488.743,Z 450.108,A -85,B 0,C 180,E1 -6398.268,E2 -6398.268} C_VEL
LIN {X 0,Y 488.767,Z 450.104,A -85,B 0,C 180,E1 -6401.613,E2 -6401.613} C_VEL
LIN {X 0,Y 488.731,Z 450.105,A -85,B 0,C 180,E1 -6405.001,E2 -6405.001} C_VEL
LIN {X 0,Y 488.727,Z 450.108,A -85,B 0,C 180,E1 -6408.443,E2 -6408.443} C_VEL
LIN {X 0,Y 488.689,Z 450.109,A -85,B 0,C 180,E1 -6411.071,E2 -6411.071} C_VEL
LIN {X 0,Y 488.652,Z 450.119,A -85,B 0,C 180,E1 -6413.747,E2 -6413.747} C_VEL
LIN {X 0,Y 488.68,Z 450.11,A -85,B 0,C 180,E1 -6416.922,E2 -6416.922} C_VEL
LIN {X 0,Y 488.699,Z 450.109,A -85,B 0,C 180,E1 -6420.221,E2 -6420.221} C_VEL
LIN {X 0,Y 488.691,Z 450.108,A -85,B 0,C 180,E1 -6423.48,E2 -6423.48} C_VEL
LIN {X 0,Y 488.633,Z 450.118,A -85,B 0,C 180,E1 -6426.35,E2 -6426.35} C_VEL
LIN {X 0,Y 488.656,Z 450.112,A -85,B 0,C 180,E1 -6429.258,E2 -6429.258} C_VEL
LIN {X 0,Y 488.633,Z 450.103,A -85,B 0,C 180,E1 -6432.531,E2 -6432.531} C_VEL
LIN {X 0,Y 488.685,Z 450.106,A -85,B 0,C 180,E1 -6435.198,E2 -6435.198} C_VEL
LIN {X 0,Y 488.647,Z 450.108,A -85,B 0,C 180,E1 -6438.581,E2 -6438.581} C_VEL
LIN {X 0,Y 488.674,Z 450.108,A -85,B 0,C 180,E1 -6440.951,E2 -6440.951} C_VEL
LIN {X 0,Y 488.632,Z 450.119,A -85,B 0,C 180,E1 -6443.866,E2 -6443.866} C_VEL
LIN {X 0,Y 488.695,Z 450.106,A -85,B 0,C 180,E1 -6446.522,E2 -6446.522} C_VEL
LIN {X 0,Y 488.704,Z 450.112,A -85,B 0,C 180,E1 -6449.781,E2 -6449.781} C_VEL
LIN {X 0,Y 488.684,Z 450.099,A -85,B 0,C 180,E1 -6453.08,E2 -6453.08} C_VEL
LIN {X 0,Y 488.658,Z 450.115,A -85,B 0,C 180,E1 -6456.254,E2 -6456.254} C_VEL
LIN {X 0,Y 488.704,Z 450.101,A -85,B 0,C 180,E1 -6459.187,E2 -6459.187} C_VEL
LIN {X 0,Y 488.696,Z 450.099,A -85,B 0,C 180,E1 -6461.649,E2 -6461.649} C_VEL
LIN {X 0,Y 488.733,Z 450.102,A -85,B 0,C 180,E1 -6465,E2 -6465} C_VEL
LIN {X 0,Y 488.775,Z 450.089,A -85,B 0,C 180,E1 -6468.388,E2 -6468.388} C_VEL
LIN {X 0,Y 488.746,Z 450.097,A -85,B 0,C 180,E1 -6471.734,E2 -6471.734} C_VEL
LIN {X 0,Y 488.804,Z 450.097,A -85,B 0,C 180,E1 -6474.225,E2 -6474.225} C_VEL
LIN {X 0,Y 488.934,Z 450.076,A -85,B 0,C 180,E1 -6477.53,E2 -6477.53} C_VEL
LIN {X 0,Y 488.934,Z 450.07,A -85,B 0,C 180,E1 -6480.001,E2 -6480.001} C_VEL
LIN {X 0,Y 488.935,Z 450.077,A -85,B 0,C 180,E1 -6482.473,E2 -6482.473} C_VEL
LIN {X 0,Y 488.804,Z 450.099,A -85,B 0,C 180,E1 -6485.778,E2 -6485.778} C_VEL
LIN {X 0,Y 488.749,Z 450.09,A -85,B 0,C 180,E1 -6488.269,E2 -6488.269} C_VEL
LIN {X 0,Y 488.78,Z 450.093,A -85,B 0,C 180,E1 -6491.614,E2 -6491.614} C_VEL
LIN {X 0,Y 488.712,Z 450.103,A -85,B 0,C 180,E1 -6495.003,E2 -6495.003} C_VEL
LIN {X 0,Y 488.699,Z 450.096,A -85,B 0,C 180,E1 -6498.445,E2 -6498.445} C_VEL
LIN {X 0,Y 488.676,Z 450.106,A -85,B 0,C 180,E1 -6501.073,E2 -6501.073} C_VEL
LIN {X 0,Y 488.667,Z 450.116,A -85,B 0,C 180,E1 -6503.748,E2 -6503.748} C_VEL
LIN {X 0,Y 488.694,Z 450.096,A -85,B 0,C 180,E1 -6506.922,E2 -6506.922} C_VEL
LIN {X 0,Y 488.715,Z 450.108,A -85,B 0,C 180,E1 -6510.221,E2 -6510.221} C_VEL
LIN {X 0,Y 488.707,Z 450.103,A -85,B 0,C 180,E1 -6513.48,E2 -6513.48} C_VEL
LIN {X 0,Y 488.647,Z 450.116,A -85,B 0,C 180,E1 -6516.35,E2 -6516.35} C_VEL
LIN {X 0,Y 488.668,Z 450.108,A -85,B 0,C 180,E1 -6519.258,E2 -6519.258} C_VEL
LIN {X 0,Y 488.647,Z 450.113,A -85,B 0,C 180,E1 -6522.531,E2 -6522.531} C_VEL
LIN {X 0,Y 488.696,Z 450.107,A -85,B 0,C 180,E1 -6525.197,E2 -6525.197} C_VEL
LIN {X 0,Y 488.643,Z 450.104,A -85,B 0,C 180,E1 -6528.578,E2 -6528.578} C_VEL
LIN {X 0,Y 488.653,Z 450.119,A -85,B 0,C 180,E1 -6531.798,E2 -6531.798} C_VEL
LIN {X 0,Y 488.703,Z 450.106,A -85,B 0,C 180,E1 -6535.057,E2 -6535.057} C_VEL
LIN {X 0,Y 488.691,Z 450.114,A -85,B 0,C 180,E1 -6538.05,E2 -6538.05} C_VEL
LIN {X 0,Y 488.686,Z 450.112,A -85,B 0,C 180,E1 -6540.728,E2 -6540.728} C_VEL
LIN {X 0,Y 488.75,Z 450.319,A -85,B 0,C 180,E1 -6543.068,E2 -6543.068} C_VEL
LIN {X 0,Y 490.264,Z 458.768,A -85,B 0,C 180,E1 -6545.047,E2 -6545.047} C_VEL
LIN {X 0,Y 490.171,Z 465.811,A -85,B 0,C 180,E1 -6546.582,E2 -6546.582} C_VEL
LIN {X 0,Y 489.625,Z 480.297,A -85,B 0,C 180,E1 -6549.63,E2 -6549.63} C_VEL
LIN {X 0,Y 489.155,Z 493.726,A -85,B 0,C 180,E1 -6552.439,E2 -6552.439} C_VEL
LIN {X 0,Y 488.99,Z 499.938,A -85,B 0,C 180,E1 -6553.714,E2 -6553.714} C_VEL
LIN {X 0,Y 490.71,Z 510.184,A -85,B 0,C 180,E1 -6553.954,E2 -6553.954} C_VEL
LIN {X 0,Y 491.691,Z 516.512,A -85,B 0,C 180,E1 -6554.081,E2 -6554.081} C_VEL
LIN {X 0,Y 491.147,Z 604.766,A -85,B 0,C 180,E1 -6555.392,E2 -6555.392} C_VEL
LIN {X 0,Y 490.952,Z 614.685,A -85,B 0,C 180,E1 -6555.625,E2 -6555.625} C_VEL
LIN {X 0,Y 490.681,Z 624.675,A -85,B 0,C 180,E1 -6555.96,E2 -6555.96} C_VEL
LIN {X 0,Y 490.344,Z 635.035,A -85,B 0,C 180,E1 -6556.426,E2 -6556.426} C_VEL
LIN {X 0,Y 490.046,Z 644.326,A -85,B 0,C 180,E1 -6556.955,E2 -6556.955} C_VEL
LIN {X 0,Y 489.749,Z 653.192,A -85,B 0,C 180,E1 -6557.57,E2 -6557.57} C_VEL
LIN {X 0,Y 489.459,Z 661.924,A -85,B 0,C 180,E1 -6558.298,E2 -6558.298} C_VEL
LIN {X 0,Y 489.121,Z 669.347,A -85,B 0,C 180,E1 -6559.025,E2 -6559.025} C_VEL
LIN {X 0,Y 488.722,Z 678.145,A -85,B 0,C 180,E1 -6560.063,E2 -6560.063} C_VEL
LIN {X 0,Y 488.525,Z 684.137,A -85,B 0,C 180,E1 -6560.895,E2 -6560.895} C_VEL
LIN {X 0,Y 488.326,Z 690.449,A -85,B 0,C 180,E1 -6561.934,E2 -6561.934} C_VEL
LIN {X 0,Y 488.182,Z 695.723,A -85,B 0,C 180,E1 -6562.971,E2 -6562.971} C_VEL
LIN {X 0,Y 488.028,Z 700.813,A -85,B 0,C 180,E1 -6564.215,E2 -6564.215} C_VEL
LIN {X 0,Y 487.922,Z 704.772,A -85,B 0,C 180,E1 -6565.456,E2 -6565.456} C_VEL
LIN {X 0,Y 487.965,Z 707.703,A -85,B 0,C 180,E1 -6566.697,E2 -6566.697} C_VEL
LIN {X 0,Y 487.91,Z 709.199,A -85,B 0,C 180,E1 -6567.523,E2 -6567.523} C_VEL
LIN {X 0,Y 487.834,Z 710.716,A -85,B 0,C 180,E1 -6569.175,E2 -6569.175} C_VEL
LIN {X 0,Y 487.819,Z 710.994,A -85,B 0,C 180,E1 -6570,E2 -6570} C_VEL
LIN {X 0,Y 487.891,Z 710.124,A -85,B 0,C 180,E1 -6571.651,E2 -6571.651} C_VEL
LIN {X 0,Y 487.91,Z 709.199,A -85,B 0,C 180,E1 -6572.477,E2 -6572.477} C_VEL
LIN {X 0,Y 487.928,Z 705.86,A -85,B 0,C 180,E1 -6574.13,E2 -6574.13} C_VEL
LIN {X 0,Y 488.022,Z 702.24,A -85,B 0,C 180,E1 -6575.371,E2 -6575.371} C_VEL
LIN {X 0,Y 488.07,Z 697.51,A -85,B 0,C 180,E1 -6576.615,E2 -6576.615} C_VEL
LIN {X 0,Y 488.252,Z 691.541,A -85,B 0,C 180,E1 -6577.859,E2 -6577.859} C_VEL
LIN {X 0,Y 488.466,Z 685.449,A -85,B 0,C 180,E1 -6578.898,E2 -6578.898} C_VEL
LIN {X 0,Y 488.687,Z 679.707,A -85,B 0,C 180,E1 -6579.728,E2 -6579.728} C_VEL
LIN {X 0,Y 488.942,Z 673.049,A -85,B 0,C 180,E1 -6580.56,E2 -6580.56} C_VEL
LIN {X 0,Y 489.269,Z 665.219,A -85,B 0,C 180,E1 -6581.391,E2 -6581.391} C_VEL
LIN {X 0,Y 489.655,Z 657.134,A -85,B 0,C 180,E1 -6582.117,E2 -6582.117} C_VEL
LIN {X 0,Y 489.96,Z 647.51,A -85,B 0,C 180,E1 -6582.836,E2 -6582.836} C_VEL
LIN {X 0,Y 490.235,Z 638.973,A -85,B 0,C 180,E1 -6583.366,E2 -6583.366} C_VEL
LIN {X 0,Y 490.609,Z 628.465,A -85,B 0,C 180,E1 -6583.883,E2 -6583.883} C_VEL
LIN {X 0,Y 490.922,Z 618.131,A -85,B 0,C 180,E1 -6584.27,E2 -6584.27} C_VEL
LIN {X 0,Y 491.035,Z 607.408,A -85,B 0,C 180,E1 -6584.558,E2 -6584.558} C_VEL
LIN {X 0,Y 491.29,Z 588.215,A -85,B 0,C 180,E1 -6584.868,E2 -6584.868} C_VEL
LIN {X 0,Y 491.545,Z 515.199,A -85,B 0,C 180,E1 -6585.943,E2 -6585.943} C_VEL
LIN {X 0,Y 488.961,Z 500.065,A -85,B 0,C 180,E1 -6586.277,E2 -6586.277} C_VEL
LIN {X 0,Y 488.945,Z 499.259,A -85,B 0,C 180,E1 -6586.385,E2 -6586.385} C_VEL
LIN {X 0,Y 489.435,Z 486.565,A -85,B 0,C 180,E1 -6589.076,E2 -6589.076} C_VEL
LIN {X 0,Y 489.902,Z 471.959,A -85,B 0,C 180,E1 -6592.121,E2 -6592.121} C_VEL
LIN {X 0,Y 490.368,Z 460.576,A -85,B 0,C 180,E1 -6594.559,E2 -6594.559} C_VEL
LIN {X 0,Y 489.52,Z 454.38,A -85,B 0,C 180,E1 -6595.969,E2 -6595.969} C_VEL
LIN {X 0,Y 488.729,Z 450.22,A -85,B 0,C 180,E1 -6596.98,E2 -6596.98} C_VEL
LIN {X 0,Y 488.691,Z 450.111,A -85,B 0,C 180,E1 -6600.358,E2 -6600.358} C_VEL
LIN {X 0,Y 488.711,Z 450.104,A -85,B 0,C 180,E1 -6603.479,E2 -6603.479} C_VEL
LIN {X 0,Y 488.648,Z 450.113,A -85,B 0,C 180,E1 -6606.348,E2 -6606.348} C_VEL
LIN {X 0,Y 488.672,Z 450.109,A -85,B 0,C 180,E1 -6609.256,E2 -6609.256} C_VEL
LIN {X 0,Y 488.649,Z 450.115,A -85,B 0,C 180,E1 -6612.53,E2 -6612.53} C_VEL
LIN {X 0,Y 488.696,Z 450.105,A -85,B 0,C 180,E1 -6615.196,E2 -6615.196} C_VEL
LIN {X 0,Y 488.642,Z 450.114,A -85,B 0,C 180,E1 -6618.577,E2 -6618.577} C_VEL
LIN {X 0,Y 488.648,Z 450.114,A -85,B 0,C 180,E1 -6621.796,E2 -6621.796} C_VEL
LIN {X 0,Y 488.712,Z 450.1,A -85,B 0,C 180,E1 -6625.054,E2 -6625.054} C_VEL
LIN {X 0,Y 488.691,Z 450.111,A -85,B 0,C 180,E1 -6628.047,E2 -6628.047} C_VEL
LIN {X 0,Y 488.697,Z 450.106,A -85,B 0,C 180,E1 -6630.727,E2 -6630.727} C_VEL
LIN {X 0,Y 488.677,Z 450.1,A -85,B 0,C 180,E1 -6633.522,E2 -6633.522} C_VEL
LIN {X 0,Y 488.667,Z 450.116,A -85,B 0,C 180,E1 -6636.252,E2 -6636.252} C_VEL
LIN {X 0,Y 488.67,Z 450.106,A -85,B 0,C 180,E1 -6639.198,E2 -6639.198} C_VEL
LIN {X 0,Y 488.656,Z 450.108,A -85,B 0,C 180,E1 -6642.419,E2 -6642.419} C_VEL
LIN {X 0,Y 488.712,Z 450.103,A -85,B 0,C 180,E1 -6644.997,E2 -6644.997} C_VEL
LIN {X 0,Y 488.78,Z 450.093,A -85,B 0,C 180,E1 -6648.386,E2 -6648.386} C_VEL
LIN {X 0,Y 488.749,Z 450.09,A -85,B 0,C 180,E1 -6651.731,E2 -6651.731} C_VEL
LIN {X 0,Y 488.804,Z 450.099,A -85,B 0,C 180,E1 -6654.222,E2 -6654.222} C_VEL
LIN {X 0,Y 488.935,Z 450.077,A -85,B 0,C 180,E1 -6657.527,E2 -6657.527} C_VEL
LIN {X 0,Y 488.935,Z 450.07,A -85,B 0,C 180,E1 -6659.999,E2 -6659.999} C_VEL
LIN {X 0,Y 488.934,Z 450.076,A -85,B 0,C 180,E1 -6662.47,E2 -6662.47} C_VEL
LIN {X 0,Y 488.804,Z 450.097,A -85,B 0,C 180,E1 -6665.775,E2 -6665.775} C_VEL
LIN {X 0,Y 488.746,Z 450.097,A -85,B 0,C 180,E1 -6668.266,E2 -6668.266} C_VEL
LIN {X 0,Y 488.775,Z 450.089,A -85,B 0,C 180,E1 -6671.612,E2 -6671.612} C_VEL
LIN {X 0,Y 488.733,Z 450.102,A -85,B 0,C 180,E1 -6675,E2 -6675} C_VEL
LIN {X 0,Y 488.694,Z 450.098,A -85,B 0,C 180,E1 -6678.443,E2 -6678.443} C_VEL
LIN {X 0,Y 488.691,Z 450.102,A -85,B 0,C 180,E1 -6681.07,E2 -6681.07} C_VEL
LIN {X 0,Y 488.658,Z 450.115,A -85,B 0,C 180,E1 -6683.746,E2 -6683.746} C_VEL
LIN {X 0,Y 488.684,Z 450.099,A -85,B 0,C 180,E1 -6686.92,E2 -6686.92} C_VEL
LIN {X 0,Y 488.704,Z 450.112,A -85,B 0,C 180,E1 -6690.219,E2 -6690.219} C_VEL
LIN {X 0,Y 488.695,Z 450.106,A -85,B 0,C 180,E1 -6693.478,E2 -6693.478} C_VEL
LIN {X 0,Y 488.635,Z 450.119,A -85,B 0,C 180,E1 -6696.348,E2 -6696.348} C_VEL
LIN {X 0,Y 488.673,Z 450.109,A -85,B 0,C 180,E1 -6699.255,E2 -6699.255} C_VEL
LIN {X 0,Y 488.653,Z 450.109,A -85,B 0,C 180,E1 -6701.593,E2 -6701.593} C_VEL
LIN {X 0,Y 488.685,Z 450.106,A -85,B 0,C 180,E1 -6704.802,E2 -6704.802} C_VEL
LIN {X 0,Y 488.633,Z 450.103,A -85,B 0,C 180,E1 -6707.469,E2 -6707.469} C_VEL
LIN {X 0,Y 488.656,Z 450.112,A -85,B 0,C 180,E1 -6710.742,E2 -6710.742} C_VEL
LIN {X 0,Y 488.629,Z 450.116,A -85,B 0,C 180,E1 -6713.864,E2 -6713.864} C_VEL
LIN {X 0,Y 488.691,Z 450.108,A -85,B 0,C 180,E1 -6716.52,E2 -6716.52} C_VEL
LIN {X 0,Y 488.699,Z 450.109,A -85,B 0,C 180,E1 -6719.779,E2 -6719.779} C_VEL
LIN {X 0,Y 488.68,Z 450.11,A -85,B 0,C 180,E1 -6723.078,E2 -6723.078} C_VEL
LIN {X 0,Y 488.664,Z 450.114,A -85,B 0,C 180,E1 -6724.311,E2 -6724.311} C_VEL
LIN {X 0,Y 488.032,Z 450.197,A -85,B 0,C 180,E1 -6724.999,E2 -6724.999} C_VEL
LIN {X 0,Y 485.189,Z 450.555,A -85,B 0,C 180,E1 -6726.117,E2 -6726.117} C_VEL
LIN {X 0,Y 482.759,Z 450.855,A -85,B 0,C 180,E1 -6727.017,E2 -6727.017} C_VEL
LIN {X 0,Y 481.706,Z 450.983,A -85,B 0,C 180,E1 -6727.713,E2 -6727.713} C_VEL
LIN {X 0,Y 481.617,Z 450.992,A -85,B 0,C 180,E1 -6727.948,E2 -6727.948} C_VEL
LIN {X 0,Y 481.679,Z 450.987,A -85,B 0,C 180,E1 -6730.392,E2 -6730.392} C_VEL
LIN {X 0,Y 481.601,Z 450.993,A -85,B 0,C 180,E1 -6733.031,E2 -6733.031} C_VEL
LIN {X 0,Y 481.659,Z 450.989,A -85,B 0,C 180,E1 -6735.638,E2 -6735.638} C_VEL
LIN {X 0,Y 481.718,Z 450.983,A -85,B 0,C 180,E1 -6738.214,E2 -6738.214} C_VEL
LIN {X 0,Y 481.702,Z 450.984,A -85,B 0,C 180,E1 -6741.611,E2 -6741.611} C_VEL
LIN {X 0,Y 481.757,Z 450.979,A -85,B 0,C 180,E1 -6744.139,E2 -6744.139} C_VEL
LIN {X 0,Y 481.89,Z 450.96,A -85,B 0,C 180,E1 -6747.492,E2 -6747.492} C_VEL
LIN {X 0,Y 481.893,Z 450.962,A -85,B 0,C 180,E1 -6750,E2 -6750} C_VEL
LIN {X 0,Y 481.89,Z 450.96,A -85,B 0,C 180,E1 -6752.508,E2 -6752.508} C_VEL
LIN {X 0,Y 481.757,Z 450.979,A -85,B 0,C 180,E1 -6755.861,E2 -6755.861} C_VEL
LIN {X 0,Y 481.702,Z 450.984,A -85,B 0,C 180,E1 -6758.389,E2 -6758.389} C_VEL
LIN {X 0,Y 481.718,Z 450.983,A -85,B 0,C 180,E1 -6761.786,E2 -6761.786} C_VEL
LIN {X 0,Y 481.713,Z 450.98,A -85,B 0,C 180,E1 -6765.225,E2 -6765.225} C_VEL
LIN {X 0,Y 481.688,Z 450.983,A -85,B 0,C 180,E1 -6768.722,E2 -6768.722} C_VEL
LIN {X 0,Y 481.627,Z 450.991,A -85,B 0,C 180,E1 -6771.395,E2 -6771.395} C_VEL
LIN {X 0,Y 481.631,Z 450.994,A -85,B 0,C 180,E1 -6774.115,E2 -6774.115} C_VEL
LIN {X 0,Y 481.635,Z 450.988,A -85,B 0,C 180,E1 -6777.117,E2 -6777.117} C_VEL
LIN {X 0,Y 481.648,Z 450.98,A -85,B 0,C 180,E1 -6779.743,E2 -6779.743} C_VEL
LIN {X 0,Y 481.631,Z 450.986,A -85,B 0,C 180,E1 -6782.677,E2 -6782.677} C_VEL
LIN {X 0,Y 481.633,Z 450.975,A -85,B 0,C 180,E1 -6785.202,E2 -6785.202} C_VEL
LIN {X 0,Y 481.613,Z 450.997,A -85,B 0,C 180,E1 -6788.004,E2 -6788.004} C_VEL
LIN {X 0,Y 481.588,Z 450.98,A -85,B 0,C 180,E1 -6791.048,E2 -6791.048} C_VEL
LIN {X 0,Y 481.636,Z 450.986,A -85,B 0,C 180,E1 -6794.46,E2 -6794.46} C_VEL
LIN {X 0,Y 481.601,Z 450.991,A -85,B 0,C 180,E1 -6796.856,E2 -6796.856} C_VEL
LIN {X 0,Y 481.642,Z 450.988,A -85,B 0,C 180,E1 -6800.058,E2 -6800.058} C_VEL
LIN {X 0,Y 481.593,Z 450.993,A -85,B 0,C 180,E1 -6803.381,E2 -6803.381} C_VEL
LIN {X 0,Y 481.658,Z 450.984,A -85,B 0,C 180,E1 -6806.328,E2 -6806.328} C_VEL
LIN {X 0,Y 481.629,Z 450.989,A -85,B 0,C 180,E1 -6809.421,E2 -6809.421} C_VEL
LIN {X 0,Y 481.636,Z 450.981,A -85,B 0,C 180,E1 -6812.166,E2 -6812.166} C_VEL
LIN {X 0,Y 481.66,Z 450.981,A -85,B 0,C 180,E1 -6814.968,E2 -6814.968} C_VEL
LIN {X 0,Y 481.635,Z 450.991,A -85,B 0,C 180,E1 -6817.706,E2 -6817.706} C_VEL
LIN {X 0,Y 481.638,Z 450.975,A -85,B 0,C 180,E1 -6820.392,E2 -6820.392} C_VEL
LIN {X 0,Y 481.6,Z 450.987,A -85,B 0,C 180,E1 -6823.032,E2 -6823.032} C_VEL
LIN {X 0,Y 481.66,Z 450.987,A -85,B 0,C 180,E1 -6825.639,E2 -6825.639} C_VEL
LIN {X 0,Y 481.726,Z 450.969,A -85,B 0,C 180,E1 -6828.216,E2 -6828.216} C_VEL
LIN {X 0,Y 481.704,Z 450.972,A -85,B 0,C 180,E1 -6831.612,E2 -6831.612} C_VEL
LIN {X 0,Y 481.766,Z 450.975,A -85,B 0,C 180,E1 -6834.14,E2 -6834.14} C_VEL
LIN {X 0,Y 481.899,Z 450.952,A -85,B 0,C 180,E1 -6837.494,E2 -6837.494} C_VEL
LIN {X 0,Y 481.904,Z 450.945,A -85,B 0,C 180,E1 -6840.001,E2 -6840.001} C_VEL
LIN {X 0,Y 481.9,Z 450.953,A -85,B 0,C 180,E1 -6842.509,E2 -6842.509} C_VEL
LIN {X 0,Y 481.766,Z 450.976,A -85,B 0,C 180,E1 -6845.862,E2 -6845.862} C_VEL
LIN {X 0,Y 481.707,Z 450.965,A -85,B 0,C 180,E1 -6848.39,E2 -6848.39} C_VEL
LIN {X 0,Y 481.731,Z 450.973,A -85,B 0,C 180,E1 -6851.787,E2 -6851.787} C_VEL
LIN {X 0,Y 481.687,Z 450.979,A -85,B 0,C 180,E1 -6855.227,E2 -6855.227} C_VEL
LIN {X 0,Y 481.632,Z 450.974,A -85,B 0,C 180,E1 -6858.726,E2 -6858.726} C_VEL
LIN {X 0,Y 481.621,Z 450.986,A -85,B 0,C 180,E1 -6861.397,E2 -6861.397} C_VEL
LIN {X 0,Y 481.645,Z 450.986,A -85,B 0,C 180,E1 -6864.116,E2 -6864.116} C_VEL
LIN {X 0,Y 481.649,Z 450.974,A -85,B 0,C 180,E1 -6867.117,E2 -6867.117} C_VEL
LIN {X 0,Y 481.663,Z 450.987,A -85,B 0,C 180,E1 -6869.743,E2 -6869.743} C_VEL
LIN {X 0,Y 481.646,Z 450.98,A -85,B 0,C 180,E1 -6872.677,E2 -6872.677} C_VEL
LIN {X 0,Y 481.648,Z 450.981,A -85,B 0,C 180,E1 -6875.203,E2 -6875.203} C_VEL
LIN {X 0,Y 481.625,Z 450.992,A -85,B 0,C 180,E1 -6878.003,E2 -6878.003} C_VEL
LIN {X 0,Y 481.603,Z 450.989,A -85,B 0,C 180,E1 -6881.048,E2 -6881.048} C_VEL
LIN {X 0,Y 481.65,Z 450.985,A -85,B 0,C 180,E1 -6884.46,E2 -6884.46} C_VEL
LIN {X 0,Y 481.613,Z 450.989,A -85,B 0,C 180,E1 -6886.857,E2 -6886.857} C_VEL
LIN {X 0,Y 481.63,Z 450.986,A -85,B 0,C 180,E1 -6890.055,E2 -6890.055} C_VEL
LIN {X 0,Y 481.605,Z 450.99,A -85,B 0,C 180,E1 -6893.252,E2 -6893.252} C_VEL
LIN {X 0,Y 481.673,Z 450.982,A -85,B 0,C 180,E1 -6896.328,E2 -6896.328} C_VEL
LIN {X 0,Y 481.634,Z 450.991,A -85,B 0,C 180,E1 -6899.422,E2 -6899.422} C_VEL
LIN {X 0,Y 481.701,Z 451.096,A -85,B 0,C 180,E1 -6902.817,E2 -6902.817} C_VEL
LIN {X 0,Y 483.34,Z 460.424,A -85,B 0,C 180,E1 -6905.06,E2 -6905.06} C_VEL
LIN {X 0,Y 483.107,Z 468.677,A -85,B 0,C 180,E1 -6906.873,E2 -6906.873} C_VEL
LIN {X 0,Y 482.57,Z 482.191,A -85,B 0,C 180,E1 -6909.764,E2 -6909.764} C_VEL
LIN {X 0,Y 482.086,Z 495.618,A -85,B 0,C 180,E1 -6912.611,E2 -6912.611} C_VEL
LIN {X 0,Y 481.986,Z 499.747,A -85,B 0,C 180,E1 -6913.47,E2 -6913.47} C_VEL
LIN {X 0,Y 483.638,Z 509.698,A -85,B 0,C 180,E1 -6913.709,E2 -6913.709} C_VEL
LIN {X 0,Y 484.877,Z 517.732,A -85,B 0,C 180,E1 -6913.873,E2 -6913.873} C_VEL
LIN {X 0,Y 484.294,Z 604.57,A -85,B 0,C 180,E1 -6915.181,E2 -6915.181} C_VEL
LIN {X 0,Y 484.077,Z 614.489,A -85,B 0,C 180,E1 -6915.416,E2 -6915.416} C_VEL
LIN {X 0,Y 483.775,Z 624.478,A -85,B 0,C 180,E1 -6915.756,E2 -6915.756} C_VEL
LIN {X 0,Y 483.452,Z 634.839,A -85,B 0,C 180,E1 -6916.229,E2 -6916.229} C_VEL
LIN {X 0,Y 483.125,Z 643.992,A -85,B 0,C 180,E1 -6916.755,E2 -6916.755} C_VEL
LIN {X 0,Y 482.787,Z 652.995,A -85,B 0,C 180,E1 -6917.388,E2 -6917.388} C_VEL
LIN {X 0,Y 482.485,Z 661.727,A -85,B 0,C 180,E1 -6918.127,E2 -6918.127} C_VEL
LIN {X 0,Y 482.133,Z 669.151,A -85,B 0,C 180,E1 -6918.864,E2 -6918.864} C_VEL
LIN {X 0,Y 481.691,Z 677.948,A -85,B 0,C 180,E1 -6919.917,E2 -6919.917} C_VEL
LIN {X 0,Y 481.467,Z 683.94,A -85,B 0,C 180,E1 -6920.76,E2 -6920.76} C_VEL
LIN {X 0,Y 481.257,Z 690.252,A -85,B 0,C 180,E1 -6921.814,E2 -6921.814} C_VEL
LIN {X 0,Y 481.1,Z 695.525,A -85,B 0,C 180,E1 -6922.867,E2 -6922.867} C_VEL
LIN {X 0,Y 480.932,Z 700.616,A -85,B 0,C 180,E1 -6924.129,E2 -6924.129} C_VEL
LIN {X 0,Y 480.84,Z 704.576,A -85,B 0,C 180,E1 -6925.389,E2 -6925.389} C_VEL
LIN {X 0,Y 480.889,Z 707.507,A -85,B 0,C 180,E1 -6926.649,E2 -6926.649} C_VEL
LIN {X 0,Y 480.824,Z 709.003,A -85,B 0,C 180,E1 -6927.487,E2 -6927.487} C_VEL
LIN {X 0,Y 480.76,Z 710.52,A -85,B 0,C 180,E1 -6929.162,E2 -6929.162} C_VEL
LIN {X 0,Y 480.743,Z 710.798,A -85,B 0,C 180,E1 -6930,E2 -6930} C_VEL
LIN {X 0,Y 480.793,Z 709.927,A -85,B 0,C 180,E1 -6931.675,E2 -6931.675} C_VEL
LIN {X 0,Y 480.824,Z 709.003,A -85,B 0,C 180,E1 -6932.513,E2 -6932.513} C_VEL
LIN {X 0,Y 480.889,Z 707.507,A -85,B 0,C 180,E1 -6933.351,E2 -6933.351} C_VEL
LIN {X 0,Y 480.899,Z 703.454,A -85,B 0,C 180,E1 -6935.03,E2 -6935.03} C_VEL
LIN {X 0,Y 480.952,Z 698.432,A -85,B 0,C 180,E1 -6936.45,E2 -6936.45} C_VEL
LIN {X 0,Y 481.158,Z 692.436,A -85,B 0,C 180,E1 -6937.765,E2 -6937.765} C_VEL
LIN {X 0,Y 481.382,Z 686.564,A -85,B 0,C 180,E1 -6938.818,E2 -6938.818} C_VEL
LIN {X 0,Y 481.589,Z 681.071,A -85,B 0,C 180,E1 -6939.661,E2 -6939.661} C_VEL
LIN {X 0,Y 481.917,Z 672.851,A -85,B 0,C 180,E1 -6940.716,E2 -6940.716} C_VEL
LIN {X 0,Y 482.302,Z 665.023,A -85,B 0,C 180,E1 -6941.558,E2 -6941.558} C_VEL
LIN {X 0,Y 482.683,Z 656.937,A -85,B 0,C 180,E1 -6942.295,E2 -6942.295} C_VEL
LIN {X 0,Y 483.01,Z 647.176,A -85,B 0,C 180,E1 -6943.034,E2 -6943.034} C_VEL
LIN {X 0,Y 483.313,Z 638.777,A -85,B 0,C 180,E1 -6943.561,E2 -6943.561} C_VEL
LIN {X 0,Y 483.699,Z 628.268,A -85,B 0,C 180,E1 -6944.086,E2 -6944.086} C_VEL
LIN {X 0,Y 484.03,Z 617.935,A -85,B 0,C 180,E1 -6944.478,E2 -6944.478} C_VEL
LIN {X 0,Y 484.175,Z 607.212,A -85,B 0,C 180,E1 -6944.769,E2 -6944.769} C_VEL
LIN {X 0,Y 484.45,Z 588.019,A -85,B 0,C 180,E1 -6945.083,E2 -6945.083} C_VEL
LIN {X 0,Y 484.734,Z 516.187,A -85,B 0,C 180,E1 -6946.156,E2 -6946.156} C_VEL
LIN {X 0,Y 481.958,Z 499.918,A -85,B 0,C 180,E1 -6946.518,E2 -6946.518} C_VEL
LIN {X 0,Y 481.951,Z 499.062,A -85,B 0,C 180,E1 -6946.629,E2 -6946.629} C_VEL
LIN {X 0,Y 482.453,Z 486.562,A -85,B 0,C 180,E1 -6949.332,E2 -6949.332} C_VEL
LIN {X 0,Y 482.919,Z 472.867,A -85,B 0,C 180,E1 -6952.233,E2 -6952.233} C_VEL
LIN {X 0,Y 483.404,Z 461.474,A -85,B 0,C 180,E1 -6954.707,E2 -6954.707} C_VEL
LIN {X 0,Y 482.288,Z 454.264,A -85,B 0,C 180,E1 -6956.388,E2 -6956.388} C_VEL
LIN {X 0,Y 481.701,Z 451.091,A -85,B 0,C 180,E1 -6957.183,E2 -6957.183} C_VEL
LIN {X 0,Y 481.634,Z 450.991,A -85,B 0,C 180,E1 -6960.578,E2 -6960.578} C_VEL
LIN {X 0,Y 481.678,Z 450.983,A -85,B 0,C 180,E1 -6963.728,E2 -6963.728} C_VEL
LIN {X 0,Y 481.606,Z 450.99,A -85,B 0,C 180,E1 -6966.748,E2 -6966.748} C_VEL
LIN {X 0,Y 481.63,Z 450.986,A -85,B 0,C 180,E1 -6969.945,E2 -6969.945} C_VEL
LIN {X 0,Y 481.615,Z 450.989,A -85,B 0,C 180,E1 -6973.302,E2 -6973.302} C_VEL
LIN {X 0,Y 481.648,Z 450.986,A -85,B 0,C 180,E1 -6975.641,E2 -6975.641} C_VEL
LIN {X 0,Y 481.603,Z 450.989,A -85,B 0,C 180,E1 -6978.952,E2 -6978.952} C_VEL
LIN {X 0,Y 481.625,Z 450.992,A -85,B 0,C 180,E1 -6981.997,E2 -6981.997} C_VEL
LIN {X 0,Y 481.677,Z 450.977,A -85,B 0,C 180,E1 -6985.316,E2 -6985.316} C_VEL
LIN {X 0,Y 481.633,Z 450.992,A -85,B 0,C 180,E1 -6988.31,E2 -6988.31} C_VEL
LIN {X 0,Y 481.656,Z 450.982,A -85,B 0,C 180,E1 -6991.215,E2 -6991.215} C_VEL
LIN {X 0,Y 481.624,Z 450.983,A -85,B 0,C 180,E1 -6994.037,E2 -6994.037} C_VEL
LIN {X 0,Y 481.652,Z 450.984,A -85,B 0,C 180,E1 -6996.817,E2 -6996.817} C_VEL
LIN {X 0,Y 481.615,Z 450.987,A -85,B 0,C 180,E1 -6999.498,E2 -6999.498} C_VEL
LIN {X 0,Y 481.641,Z 450.979,A -85,B 0,C 180,E1 -7002.155,E2 -7002.155} C_VEL
LIN {X 0,Y 481.687,Z 450.979,A -85,B 0,C 180,E1 -7004.773,E2 -7004.773} C_VEL
LIN {X 0,Y 481.731,Z 450.973,A -85,B 0,C 180,E1 -7008.213,E2 -7008.213} C_VEL
LIN {X 0,Y 481.707,Z 450.965,A -85,B 0,C 180,E1 -7011.61,E2 -7011.61} C_VEL
LIN {X 0,Y 481.766,Z 450.976,A -85,B 0,C 180,E1 -7014.138,E2 -7014.138} C_VEL
LIN {X 0,Y 481.9,Z 450.953,A -85,B 0,C 180,E1 -7017.491,E2 -7017.491} C_VEL
LIN {X 0,Y 481.904,Z 450.945,A -85,B 0,C 180,E1 -7019.999,E2 -7019.999} C_VEL
LIN {X 0,Y 481.899,Z 450.952,A -85,B 0,C 180,E1 -7022.506,E2 -7022.506} C_VEL
LIN {X 0,Y 481.766,Z 450.975,A -85,B 0,C 180,E1 -7025.86,E2 -7025.86} C_VEL
LIN {X 0,Y 481.704,Z 450.972,A -85,B 0,C 180,E1 -7028.388,E2 -7028.388} C_VEL
LIN {X 0,Y 481.726,Z 450.969,A -85,B 0,C 180,E1 -7031.784,E2 -7031.784} C_VEL
LIN {X 0,Y 481.713,Z 450.977,A -85,B 0,C 180,E1 -7035.224,E2 -7035.224} C_VEL
LIN {X 0,Y 481.634,Z 450.974,A -85,B 0,C 180,E1 -7038.723,E2 -7038.723} C_VEL
LIN {X 0,Y 481.63,Z 450.983,A -85,B 0,C 180,E1 -7041.394,E2 -7041.394} C_VEL
LIN {X 0,Y 481.637,Z 450.992,A -85,B 0,C 180,E1 -7044.113,E2 -7044.113} C_VEL
LIN {X 0,Y 481.639,Z 450.976,A -85,B 0,C 180,E1 -7047.115,E2 -7047.115} C_VEL
LIN {X 0,Y 481.652,Z 450.985,A -85,B 0,C 180,E1 -7049.741,E2 -7049.741} C_VEL
LIN {X 0,Y 481.635,Z 450.985,A -85,B 0,C 180,E1 -7052.675,E2 -7052.675} C_VEL
LIN {X 0,Y 481.636,Z 450.979,A -85,B 0,C 180,E1 -7055.201,E2 -7055.201} C_VEL
LIN {X 0,Y 481.617,Z 450.997,A -85,B 0,C 180,E1 -7058.002,E2 -7058.002} C_VEL
LIN {X 0,Y 481.609,Z 450.984,A -85,B 0,C 180,E1 -7061.044,E2 -7061.044} C_VEL
LIN {X 0,Y 481.639,Z 450.986,A -85,B 0,C 180,E1 -7064.457,E2 -7064.457} C_VEL
LIN {X 0,Y 481.597,Z 450.977,A -85,B 0,C 180,E1 -7066.855,E2 -7066.855} C_VEL
LIN {X 0,Y 481.613,Z 450.986,A -85,B 0,C 180,E1 -7070.054,E2 -7070.054} C_VEL
LIN {X 0,Y 481.589,Z 450.992,A -85,B 0,C 180,E1 -7073.25,E2 -7073.25} C_VEL
LIN {X 0,Y 481.655,Z 450.982,A -85,B 0,C 180,E1 -7076.326,E2 -7076.326} C_VEL
LIN {X 0,Y 481.625,Z 450.989,A -85,B 0,C 180,E1 -7079.419,E2 -7079.419} C_VEL
LIN {X 0,Y 481.631,Z 450.992,A -85,B 0,C 180,E1 -7082.164,E2 -7082.164} C_VEL
LIN {X 0,Y 481.656,Z 450.985,A -85,B 0,C 180,E1 -7084.967,E2 -7084.967} C_VEL
LIN {X 0,Y 481.617,Z 450.992,A -85,B 0,C 180,E1 -7087.948,E2 -7087.948} C_VEL
LIN {X 0,Y 480.951,Z 451.076,A -85,B 0,C 180,E1 -7088.646,E2 -7088.646} C_VEL
LIN {X 0,Y 478.131,Z 451.43,A -85,B 0,C 180,E1 -7089.781,E2 -7089.781} C_VEL
LIN {X 0,Y 475.745,Z 451.724,A -85,B 0,C 180,E1 -7090.695,E2 -7090.695} C_VEL
LIN {X 0,Y 474.712,Z 451.853,A -85,B 0,C 180,E1 -7091.401,E2 -7091.401} C_VEL
LIN {X 0,Y 474.622,Z 451.865,A -85,B 0,C 180,E1 -7091.64,E2 -7091.64} C_VEL
LIN {X 0,Y 474.671,Z 451.858,A -85,B 0,C 180,E1 -7094.544,E2 -7094.544} C_VEL
LIN {X 0,Y 474.676,Z 451.861,A -85,B 0,C 180,E1 -7098.037,E2 -7098.037} C_VEL
LIN {X 0,Y 474.677,Z 451.858,A -85,B 0,C 180,E1 -7101.486,E2 -7101.486} C_VEL
LIN {X 0,Y 474.72,Z 451.855,A -85,B 0,C 180,E1 -7104.052,E2 -7104.052} C_VEL
LIN {X 0,Y 474.855,Z 451.836,A -85,B 0,C 180,E1 -7107.455,E2 -7107.455} C_VEL
LIN {X 0,Y 474.863,Z 451.838,A -85,B 0,C 180,E1 -7110,E2 -7110} C_VEL
LIN {X 0,Y 474.855,Z 451.836,A -85,B 0,C 180,E1 -7112.545,E2 -7112.545} C_VEL
LIN {X 0,Y 474.72,Z 451.855,A -85,B 0,C 180,E1 -7115.948,E2 -7115.948} C_VEL
LIN {X 0,Y 474.677,Z 451.858,A -85,B 0,C 180,E1 -7118.514,E2 -7118.514} C_VEL
LIN {X 0,Y 474.676,Z 451.861,A -85,B 0,C 180,E1 -7121.963,E2 -7121.963} C_VEL
LIN {X 0,Y 474.671,Z 451.859,A -85,B 0,C 180,E1 -7125.456,E2 -7125.456} C_VEL
LIN {X 0,Y 474.642,Z 451.86,A -85,B 0,C 180,E1 -7129.011,E2 -7129.011} C_VEL
LIN {X 0,Y 474.57,Z 451.873,A -85,B 0,C 180,E1 -7131.73,E2 -7131.73} C_VEL
LIN {X 0,Y 474.609,Z 451.866,A -85,B 0,C 180,E1 -7134.495,E2 -7134.495} C_VEL
LIN {X 0,Y 474.581,Z 451.868,A -85,B 0,C 180,E1 -7137.327,E2 -7137.327} C_VEL
LIN {X 0,Y 474.578,Z 451.867,A -85,B 0,C 180,E1 -7140.232,E2 -7140.232} C_VEL
LIN {X 0,Y 474.597,Z 451.862,A -85,B 0,C 180,E1 -7143.223,E2 -7143.223} C_VEL
LIN {X 0,Y 474.554,Z 451.872,A -85,B 0,C 180,E1 -7146.326,E2 -7146.326} C_VEL
LIN {X 0,Y 474.584,Z 451.867,A -85,B 0,C 180,E1 -7149.551,E2 -7149.551} C_VEL
LIN {X 0,Y 474.55,Z 451.854,A -85,B 0,C 180,E1 -7152.941,E2 -7152.941} C_VEL
LIN {X 0,Y 474.587,Z 451.869,A -85,B 0,C 180,E1 -7155.895,E2 -7155.895} C_VEL
LIN {X 0,Y 474.577,Z 451.861,A -85,B 0,C 180,E1 -7159.34,E2 -7159.34} C_VEL
LIN {X 0,Y 474.577,Z 451.87,A -85,B 0,C 180,E1 -7161.708,E2 -7161.708} C_VEL
LIN {X 0,Y 474.597,Z 451.856,A -85,B 0,C 180,E1 -7164.725,E2 -7164.725} C_VEL
LIN {X 0,Y 474.608,Z 451.865,A -85,B 0,C 180,E1 -7167.788,E2 -7167.788} C_VEL
LIN {X 0,Y 474.586,Z 451.86,A -85,B 0,C 180,E1 -7170.892,E2 -7170.892} C_VEL
LIN {X 0,Y 474.568,Z 451.86,A -85,B 0,C 180,E1 -7173.625,E2 -7173.625} C_VEL
LIN {X 0,Y 474.624,Z 451.86,A -85,B 0,C 180,E1 -7176.643,E2 -7176.643} C_VEL
LIN {X 0,Y 474.601,Z 451.854,A -85,B 0,C 180,E1 -7180.089,E2 -7180.089} C_VEL
LIN {X 0,Y 474.572,Z 451.862,A -85,B 0,C 180,E1 -7182.773,E2 -7182.773} C_VEL
LIN {X 0,Y 474.618,Z 451.862,A -85,B 0,C 180,E1 -7185.422,E2 -7185.422} C_VEL
LIN {X 0,Y 474.684,Z 451.848,A -85,B 0,C 180,E1 -7188.039,E2 -7188.039} C_VEL
LIN {X 0,Y 474.653,Z 451.848,A -85,B 0,C 180,E1 -7191.487,E2 -7191.487} C_VEL
LIN {X 0,Y 474.729,Z 451.853,A -85,B 0,C 180,E1 -7194.053,E2 -7194.053} C_VEL
LIN {X 0,Y 474.864,Z 451.828,A -85,B 0,C 180,E1 -7197.457,E2 -7197.457} C_VEL
LIN {X 0,Y 474.873,Z 451.819,A -85,B 0,C 180,E1 -7200.001,E2 -7200.001} C_VEL
LIN {X 0,Y 474.865,Z 451.829,A -85,B 0,C 180,E1 -7202.546,E2 -7202.546} C_VEL
LIN {X 0,Y 474.729,Z 451.85,A -85,B 0,C 180,E1 -7205.949,E2 -7205.949} C_VEL
LIN {X 0,Y 474.656,Z 451.842,A -85,B 0,C 180,E1 -7208.516,E2 -7208.516} C_VEL
LIN {X 0,Y 474.689,Z 451.853,A -85,B 0,C 180,E1 -7211.964,E2 -7211.964} C_VEL
LIN {X 0,Y 474.647,Z 451.857,A -85,B 0,C 180,E1 -7215.459,E2 -7215.459} C_VEL
LIN {X 0,Y 474.585,Z 451.852,A -85,B 0,C 180,E1 -7219.015,E2 -7219.015} C_VEL
LIN {X 0,Y 474.572,Z 451.868,A -85,B 0,C 180,E1 -7221.731,E2 -7221.731} C_VEL
LIN {X 0,Y 474.623,Z 451.856,A -85,B 0,C 180,E1 -7224.496,E2 -7224.496} C_VEL
LIN {X 0,Y 474.595,Z 451.853,A -85,B 0,C 180,E1 -7227.328,E2 -7227.328} C_VEL
LIN {X 0,Y 474.593,Z 451.867,A -85,B 0,C 180,E1 -7230.232,E2 -7230.232} C_VEL
LIN {X 0,Y 474.612,Z 451.857,A -85,B 0,C 180,E1 -7233.224,E2 -7233.224} C_VEL
LIN {X 0,Y 474.569,Z 451.87,A -85,B 0,C 180,E1 -7236.326,E2 -7236.326} C_VEL
LIN {X 0,Y 474.598,Z 451.864,A -85,B 0,C 180,E1 -7239.552,E2 -7239.552} C_VEL
LIN {X 0,Y 474.565,Z 451.867,A -85,B 0,C 180,E1 -7242.941,E2 -7242.941} C_VEL
LIN {X 0,Y 474.598,Z 451.871,A -85,B 0,C 180,E1 -7245.894,E2 -7245.894} C_VEL
LIN {X 0,Y 474.581,Z 451.855,A -85,B 0,C 180,E1 -7249.048,E2 -7249.048} C_VEL
LIN {X 0,Y 474.588,Z 451.87,A -85,B 0,C 180,E1 -7251.709,E2 -7251.709} C_VEL
LIN {X 0,Y 474.603,Z 451.863,A -85,B 0,C 180,E1 -7254.724,E2 -7254.724} C_VEL
LIN {X 0,Y 474.615,Z 451.863,A -85,B 0,C 180,E1 -7257.787,E2 -7257.787} C_VEL
LIN {X 0,Y 474.592,Z 451.869,A -85,B 0,C 180,E1 -7260.893,E2 -7260.893} C_VEL
LIN {X 0,Y 474.676,Z 452.106,A -85,B 0,C 180,E1 -7262.679,E2 -7262.679} C_VEL
LIN {X 0,Y 476.339,Z 461.331,A -85,B 0,C 180,E1 -7264.901,E2 -7264.901} C_VEL
LIN {X 0,Y 476.269,Z 467.047,A -85,B 0,C 180,E1 -7266.192,E2 -7266.192} C_VEL
LIN {X 0,Y 475.653,Z 480.984,A -85,B 0,C 180,E1 -7269.231,E2 -7269.231} C_VEL
LIN {X 0,Y 475.134,Z 494.415,A -85,B 0,C 180,E1 -7272.126,E2 -7272.126} C_VEL
LIN {X 0,Y 474.991,Z 499.564,A -85,B 0,C 180,E1 -7273.22,E2 -7273.22} C_VEL
LIN {X 0,Y 477.036,Z 511.729,A -85,B 0,C 180,E1 -7273.511,E2 -7273.511} C_VEL
LIN {X 0,Y 478.062,Z 518.297,A -85,B 0,C 180,E1 -7273.648,E2 -7273.648} C_VEL
LIN {X 0,Y 477.44,Z 604.374,A -85,B 0,C 180,E1 -7274.963,E2 -7274.963} C_VEL
LIN {X 0,Y 477.207,Z 614.293,A -85,B 0,C 180,E1 -7275.201,E2 -7275.201} C_VEL
LIN {X 0,Y 476.911,Z 624.282,A -85,B 0,C 180,E1 -7275.546,E2 -7275.546} C_VEL
LIN {X 0,Y 476.548,Z 634.642,A -85,B 0,C 180,E1 -7276.025,E2 -7276.025} C_VEL
LIN {X 0,Y 476.198,Z 643.795,A -85,B 0,C 180,E1 -7276.559,E2 -7276.559} C_VEL
LIN {X 0,Y 475.834,Z 652.798,A -85,B 0,C 180,E1 -7277.2,E2 -7277.2} C_VEL
LIN {X 0,Y 475.498,Z 661.567,A -85,B 0,C 180,E1 -7277.953,E2 -7277.953} C_VEL
LIN {X 0,Y 475.136,Z 668.954,A -85,B 0,C 180,E1 -7278.698,E2 -7278.698} C_VEL
LIN {X 0,Y 474.658,Z 677.75,A -85,B 0,C 180,E1 -7279.766,E2 -7279.766} C_VEL
LIN {X 0,Y 474.423,Z 683.743,A -85,B 0,C 180,E1 -7280.622,E2 -7280.622} C_VEL
LIN {X 0,Y 474.183,Z 690.054,A -85,B 0,C 180,E1 -7281.691,E2 -7281.691} C_VEL
LIN {X 0,Y 474.024,Z 695.328,A -85,B 0,C 180,E1 -7282.76,E2 -7282.76} C_VEL
LIN {X 0,Y 473.84,Z 700.419,A -85,B 0,C 180,E1 -7284.041,E2 -7284.041} C_VEL
LIN {X 0,Y 473.764,Z 704.379,A -85,B 0,C 180,E1 -7285.32,E2 -7285.32} C_VEL
LIN {X 0,Y 473.796,Z 707.311,A -85,B 0,C 180,E1 -7286.598,E2 -7286.598} C_VEL
LIN {X 0,Y 473.742,Z 708.807,A -85,B 0,C 180,E1 -7287.449,E2 -7287.449} C_VEL
LIN {X 0,Y 473.689,Z 710.325,A -85,B 0,C 180,E1 -7289.15,E2 -7289.15} C_VEL
LIN {X 0,Y 473.67,Z 710.603,A -85,B 0,C 180,E1 -7290,E2 -7290} C_VEL
LIN {X 0,Y 473.699,Z 709.731,A -85,B 0,C 180,E1 -7291.7,E2 -7291.7} C_VEL
LIN {X 0,Y 473.742,Z 708.807,A -85,B 0,C 180,E1 -7292.551,E2 -7292.551} C_VEL
LIN {X 0,Y 473.796,Z 707.311,A -85,B 0,C 180,E1 -7293.402,E2 -7293.402} C_VEL
LIN {X 0,Y 473.83,Z 703.257,A -85,B 0,C 180,E1 -7295.106,E2 -7295.106} C_VEL
LIN {X 0,Y 473.882,Z 698.629,A -85,B 0,C 180,E1 -7296.452,E2 -7296.452} C_VEL
LIN {X 0,Y 474.055,Z 693.331,A -85,B 0,C 180,E1 -7297.668,E2 -7297.668} C_VEL
LIN {X 0,Y 474.292,Z 687.679,A -85,B 0,C 180,E1 -7298.736,E2 -7298.736} C_VEL
LIN {X 0,Y 474.572,Z 680.874,A -85,B 0,C 180,E1 -7299.805,E2 -7299.805} C_VEL
LIN {X 0,Y 474.919,Z 672.654,A -85,B 0,C 180,E1 -7300.876,E2 -7300.876} C_VEL
LIN {X 0,Y 475.328,Z 664.826,A -85,B 0,C 180,E1 -7301.73,E2 -7301.73} C_VEL
LIN {X 0,Y 475.714,Z 656.825,A -85,B 0,C 180,E1 -7302.471,E2 -7302.471} C_VEL
LIN {X 0,Y 476.026,Z 648.13,A -85,B 0,C 180,E1 -7303.15,E2 -7303.15} C_VEL
LIN {X 0,Y 476.39,Z 638.58,A -85,B 0,C 180,E1 -7303.762,E2 -7303.762} C_VEL
LIN {X 0,Y 476.812,Z 628.072,A -85,B 0,C 180,E1 -7304.293,E2 -7304.293} C_VEL
LIN {X 0,Y 477.142,Z 617.738,A -85,B 0,C 180,E1 -7304.692,E2 -7304.692} C_VEL
LIN {X 0,Y 477.325,Z 607.016,A -85,B 0,C 180,E1 -7304.986,E2 -7304.986} C_VEL
LIN {X 0,Y 477.614,Z 587.823,A -85,B 0,C 180,E1 -7305.304,E2 -7305.304} C_VEL
LIN {X 0,Y 477.956,Z 517.384,A -85,B 0,C 180,E1 -7306.37,E2 -7306.37} C_VEL
LIN {X 0,Y 474.958,Z 499.738,A -85,B 0,C 180,E1 -7306.768,E2 -7306.768} C_VEL
LIN {X 0,Y 474.945,Z 498.864,A -85,B 0,C 180,E1 -7306.882,E2 -7306.882} C_VEL
LIN {X 0,Y 475.501,Z 486.294,A -85,B 0,C 180,E1 -7309.648,E2 -7309.648} C_VEL
LIN {X 0,Y 475.988,Z 472.729,A -85,B 0,C 180,E1 -7312.575,E2 -7312.575} C_VEL
LIN {X 0,Y 476.43,Z 462.355,A -85,B 0,C 180,E1 -7314.86,E2 -7314.86} C_VEL
LIN {X 0,Y 475.041,Z 454.146,A -85,B 0,C 180,E1 -7316.822,E2 -7316.822} C_VEL
LIN {X 0,Y 474.659,Z 451.978,A -85,B 0,C 180,E1 -7317.37,E2 -7317.37} C_VEL
LIN {X 0,Y 474.593,Z 451.868,A -85,B 0,C 180,E1 -7320.806,E2 -7320.806} C_VEL
LIN {X 0,Y 474.616,Z 451.859,A -85,B 0,C 180,E1 -7323.222,E2 -7323.222} C_VEL
LIN {X 0,Y 474.57,Z 451.866,A -85,B 0,C 180,E1 -7326.325,E2 -7326.325} C_VEL
LIN {X 0,Y 474.601,Z 451.864,A -85,B 0,C 180,E1 -7329.55,E2 -7329.55} C_VEL
LIN {X 0,Y 474.566,Z 451.867,A -85,B 0,C 180,E1 -7332.939,E2 -7332.939} C_VEL
LIN {X 0,Y 474.598,Z 451.865,A -85,B 0,C 180,E1 -7335.893,E2 -7335.893} C_VEL
LIN {X 0,Y 474.58,Z 451.864,A -85,B 0,C 180,E1 -7339.047,E2 -7339.047} C_VEL
LIN {X 0,Y 474.585,Z 451.865,A -85,B 0,C 180,E1 -7341.707,E2 -7341.707} C_VEL
LIN {X 0,Y 474.609,Z 451.858,A -85,B 0,C 180,E1 -7344.723,E2 -7344.723} C_VEL
LIN {X 0,Y 474.62,Z 451.859,A -85,B 0,C 180,E1 -7347.785,E2 -7347.785} C_VEL
LIN {X 0,Y 474.596,Z 451.861,A -85,B 0,C 180,E1 -7350.89,E2 -7350.89} C_VEL
LIN {X 0,Y 474.578,Z 451.856,A -85,B 0,C 180,E1 -7353.622,E2 -7353.622} C_VEL
LIN {X 0,Y 474.633,Z 451.859,A -85,B 0,C 180,E1 -7356.641,E2 -7356.641} C_VEL
LIN {X 0,Y 474.577,Z 451.861,A -85,B 0,C 180,E1 -7360.085,E2 -7360.085} C_VEL
LIN {X 0,Y 474.577,Z 451.858,A -85,B 0,C 180,E1 -7362.771,E2 -7362.771} C_VEL
LIN {X 0,Y 474.601,Z 451.861,A -85,B 0,C 180,E1 -7365.418,E2 -7365.418} C_VEL
LIN {X 0,Y 474.689,Z 451.853,A -85,B 0,C 180,E1 -7368.036,E2 -7368.036} C_VEL
LIN {X 0,Y 474.656,Z 451.842,A -85,B 0,C 180,E1 -7371.484,E2 -7371.484} C_VEL
LIN {X 0,Y 474.729,Z 451.85,A -85,B 0,C 180,E1 -7374.051,E2 -7374.051} C_VEL
LIN {X 0,Y 474.865,Z 451.829,A -85,B 0,C 180,E1 -7377.454,E2 -7377.454} C_VEL
LIN {X 0,Y 474.873,Z 451.819,A -85,B 0,C 180,E1 -7379.999,E2 -7379.999} C_VEL
LIN {X 0,Y 474.864,Z 451.828,A -85,B 0,C 180,E1 -7382.543,E2 -7382.543} C_VEL
LIN {X 0,Y 474.729,Z 451.853,A -85,B 0,C 180,E1 -7385.947,E2 -7385.947} C_VEL
LIN {X 0,Y 474.653,Z 451.848,A -85,B 0,C 180,E1 -7388.513,E2 -7388.513} C_VEL
LIN {X 0,Y 474.684,Z 451.848,A -85,B 0,C 180,E1 -7391.961,E2 -7391.961} C_VEL
LIN {X 0,Y 474.672,Z 451.855,A -85,B 0,C 180,E1 -7395.455,E2 -7395.455} C_VEL
LIN {X 0,Y 474.589,Z 451.85,A -85,B 0,C 180,E1 -7399.012,E2 -7399.012} C_VEL
LIN {X 0,Y 474.574,Z 451.865,A -85,B 0,C 180,E1 -7401.728,E2 -7401.728} C_VEL
LIN {X 0,Y 474.614,Z 451.862,A -85,B 0,C 180,E1 -7404.494,E2 -7404.494} C_VEL
LIN {X 0,Y 474.585,Z 451.855,A -85,B 0,C 180,E1 -7407.325,E2 -7407.325} C_VEL
LIN {X 0,Y 474.582,Z 451.871,A -85,B 0,C 180,E1 -7410.23,E2 -7410.23} C_VEL
LIN {X 0,Y 474.601,Z 451.86,A -85,B 0,C 180,E1 -7413.221,E2 -7413.221} C_VEL
LIN {X 0,Y 474.557,Z 451.873,A -85,B 0,C 180,E1 -7416.324,E2 -7416.324} C_VEL
LIN {X 0,Y 474.587,Z 451.867,A -85,B 0,C 180,E1 -7419.642,E2 -7419.642} C_VEL
LIN {X 0,Y 474.555,Z 451.868,A -85,B 0,C 180,E1 -7422.939,E2 -7422.939} C_VEL
LIN {X 0,Y 474.565,Z 451.864,A -85,B 0,C 180,E1 -7425.891,E2 -7425.891} C_VEL
LIN {X 0,Y 474.565,Z 451.854,A -85,B 0,C 180,E1 -7429.047,E2 -7429.047} C_VEL
LIN {X 0,Y 474.572,Z 451.87,A -85,B 0,C 180,E1 -7431.707,E2 -7431.707} C_VEL
LIN {X 0,Y 474.594,Z 451.852,A -85,B 0,C 180,E1 -7434.723,E2 -7434.723} C_VEL
LIN {X 0,Y 474.604,Z 451.866,A -85,B 0,C 180,E1 -7437.786,E2 -7437.786} C_VEL
LIN {X 0,Y 474.581,Z 451.859,A -85,B 0,C 180,E1 -7440.89,E2 -7440.89} C_VEL
LIN {X 0,Y 474.572,Z 451.871,A -85,B 0,C 180,E1 -7443.623,E2 -7443.623} C_VEL
LIN {X 0,Y 474.618,Z 451.864,A -85,B 0,C 180,E1 -7446.642,E2 -7446.642} C_VEL
LIN {X 0,Y 474.631,Z 451.866,A -85,B 0,C 180,E1 -7450.089,E2 -7450.089} C_VEL
LIN {X 0,Y 474.622,Z 451.865,A -85,B 0,C 180,E1 -7451.64,E2 -7451.64} C_VEL
LIN {X 0,Y 473.944,Z 451.953,A -85,B 0,C 180,E1 -7452.348,E2 -7452.348} C_VEL
LIN {X 0,Y 471.095,Z 452.308,A -85,B 0,C 180,E1 -7453.499,E2 -7453.499} C_VEL
LIN {X 0,Y 468.691,Z 452.604,A -85,B 0,C 180,E1 -7454.427,E2 -7454.427} C_VEL
LIN {X 0,Y 467.655,Z 452.731,A -85,B 0,C 180,E1 -7455.144,E2 -7455.144} C_VEL
LIN {X 0,Y 467.568,Z 452.742,A -85,B 0,C 180,E1 -7455.386,E2 -7455.386} C_VEL
LIN {X 0,Y 467.631,Z 452.738,A -85,B 0,C 180,E1 -7457.854,E2 -7457.854} C_VEL
LIN {X 0,Y 467.638,Z 452.734,A -85,B 0,C 180,E1 -7461.357,E2 -7461.357} C_VEL
LIN {X 0,Y 467.685,Z 452.731,A -85,B 0,C 180,E1 -7463.962,E2 -7463.962} C_VEL
LIN {X 0,Y 467.795,Z 452.715,A -85,B 0,C 180,E1 -7467.417,E2 -7467.417} C_VEL
LIN {X 0,Y 467.832,Z 452.713,A -85,B 0,C 180,E1 -7470,E2 -7470} C_VEL
LIN {X 0,Y 467.795,Z 452.715,A -85,B 0,C 180,E1 -7472.583,E2 -7472.583} C_VEL
LIN {X 0,Y 467.685,Z 452.731,A -85,B 0,C 180,E1 -7476.038,E2 -7476.038} C_VEL
LIN {X 0,Y 467.638,Z 452.734,A -85,B 0,C 180,E1 -7478.643,E2 -7478.643} C_VEL
LIN {X 0,Y 467.631,Z 452.737,A -85,B 0,C 180,E1 -7482.354,E2 -7482.354} C_VEL
LIN {X 0,Y 467.583,Z 452.744,A -85,B 0,C 180,E1 -7485.864,E2 -7485.864} C_VEL
LIN {X 0,Y 467.602,Z 452.738,A -85,B 0,C 180,E1 -7489.308,E2 -7489.308} C_VEL
LIN {X 0,Y 467.514,Z 452.753,A -85,B 0,C 180,E1 -7492.075,E2 -7492.075} C_VEL
LIN {X 0,Y 467.542,Z 452.744,A -85,B 0,C 180,E1 -7494.891,E2 -7494.891} C_VEL
LIN {X 0,Y 467.528,Z 452.75,A -85,B 0,C 180,E1 -7497.775,E2 -7497.775} C_VEL
LIN {X 0,Y 467.529,Z 452.744,A -85,B 0,C 180,E1 -7501.041,E2 -7501.041} C_VEL
LIN {X 0,Y 467.559,Z 452.729,A -85,B 0,C 180,E1 -7504.24,E2 -7504.24} C_VEL
LIN {X 0,Y 467.499,Z 452.747,A -85,B 0,C 180,E1 -7507.182,E2 -7507.182} C_VEL
LIN {X 0,Y 467.502,Z 452.738,A -85,B 0,C 180,E1 -7510.272,E2 -7510.272} C_VEL
LIN {X 0,Y 467.501,Z 452.732,A -85,B 0,C 180,E1 -7512.569,E2 -7512.569} C_VEL
LIN {X 0,Y 467.549,Z 452.738,A -85,B 0,C 180,E1 -7515.053,E2 -7515.053} C_VEL
LIN {X 0,Y 467.546,Z 452.735,A -85,B 0,C 180,E1 -7518.727,E2 -7518.727} C_VEL
LIN {X 0,Y 467.527,Z 452.752,A -85,B 0,C 180,E1 -7521.954,E2 -7521.954} C_VEL
LIN {X 0,Y 467.537,Z 452.735,A -85,B 0,C 180,E1 -7525.167,E2 -7525.167} C_VEL
LIN {X 0,Y 467.542,Z 452.747,A -85,B 0,C 180,E1 -7528.259,E2 -7528.259} C_VEL
LIN {X 0,Y 467.531,Z 452.74,A -85,B 0,C 180,E1 -7531.249,E2 -7531.249} C_VEL
LIN {X 0,Y 467.565,Z 452.74,A -85,B 0,C 180,E1 -7534.403,E2 -7534.403} C_VEL
LIN {X 0,Y 467.561,Z 452.739,A -85,B 0,C 180,E1 -7536.997,E2 -7536.997} C_VEL
LIN {X 0,Y 467.58,Z 452.732,A -85,B 0,C 180,E1 -7539.777,E2 -7539.777} C_VEL
LIN {X 0,Y 467.542,Z 452.739,A -85,B 0,C 180,E1 -7542.506,E2 -7542.506} C_VEL
LIN {X 0,Y 467.576,Z 452.738,A -85,B 0,C 180,E1 -7545.197,E2 -7545.197} C_VEL
LIN {X 0,Y 467.639,Z 452.728,A -85,B 0,C 180,E1 -7547.856,E2 -7547.856} C_VEL
LIN {X 0,Y 467.622,Z 452.722,A -85,B 0,C 180,E1 -7551.358,E2 -7551.358} C_VEL
LIN {X 0,Y 467.694,Z 452.73,A -85,B 0,C 180,E1 -7553.963,E2 -7553.963} C_VEL
LIN {X 0,Y 467.804,Z 452.707,A -85,B 0,C 180,E1 -7557.418,E2 -7557.418} C_VEL
LIN {X 0,Y 467.843,Z 452.694,A -85,B 0,C 180,E1 -7560.001,E2 -7560.001} C_VEL
LIN {X 0,Y 467.805,Z 452.708,A -85,B 0,C 180,E1 -7562.584,E2 -7562.584} C_VEL
LIN {X 0,Y 467.694,Z 452.725,A -85,B 0,C 180,E1 -7566.039,E2 -7566.039} C_VEL
LIN {X 0,Y 467.625,Z 452.716,A -85,B 0,C 180,E1 -7568.645,E2 -7568.645} C_VEL
LIN {X 0,Y 467.644,Z 452.732,A -85,B 0,C 180,E1 -7572.147,E2 -7572.147} C_VEL
LIN {X 0,Y 467.574,Z 452.741,A -85,B 0,C 180,E1 -7575.698,E2 -7575.698} C_VEL
LIN {X 0,Y 467.565,Z 452.726,A -85,B 0,C 180,E1 -7578.747,E2 -7578.747} C_VEL
LIN {X 0,Y 467.521,Z 452.75,A -85,B 0,C 180,E1 -7582.076,E2 -7582.076} C_VEL
LIN {X 0,Y 467.553,Z 452.735,A -85,B 0,C 180,E1 -7584.891,E2 -7584.891} C_VEL
LIN {X 0,Y 467.542,Z 452.736,A -85,B 0,C 180,E1 -7587.775,E2 -7587.775} C_VEL
LIN {X 0,Y 467.544,Z 452.742,A -85,B 0,C 180,E1 -7591.041,E2 -7591.041} C_VEL
LIN {X 0,Y 467.574,Z 452.736,A -85,B 0,C 180,E1 -7594.241,E2 -7594.241} C_VEL
LIN {X 0,Y 467.513,Z 452.746,A -85,B 0,C 180,E1 -7597.181,E2 -7597.181} C_VEL
LIN {X 0,Y 467.517,Z 452.747,A -85,B 0,C 180,E1 -7600.272,E2 -7600.272} C_VEL
LIN {X 0,Y 467.516,Z 452.746,A -85,B 0,C 180,E1 -7602.569,E2 -7602.569} C_VEL
LIN {X 0,Y 467.562,Z 452.739,A -85,B 0,C 180,E1 -7605.053,E2 -7605.053} C_VEL
LIN {X 0,Y 467.551,Z 452.73,A -85,B 0,C 180,E1 -7608.728,E2 -7608.728} C_VEL
LIN {X 0,Y 467.539,Z 452.749,A -85,B 0,C 180,E1 -7611.954,E2 -7611.954} C_VEL
LIN {X 0,Y 467.54,Z 452.743,A -85,B 0,C 180,E1 -7615.166,E2 -7615.166} C_VEL
LIN {X 0,Y 467.551,Z 452.748,A -85,B 0,C 180,E1 -7618.258,E2 -7618.258} C_VEL
LIN {X 0,Y 467.539,Z 452.747,A -85,B 0,C 180,E1 -7621.248,E2 -7621.248} C_VEL
LIN {X 0,Y 467.607,Z 452.988,A -85,B 0,C 180,E1 -7622.469,E2 -7622.469} C_VEL
LIN {X 0,Y 469.427,Z 463.235,A -85,B 0,C 180,E1 -7624.98,E2 -7624.98} C_VEL
LIN {X 0,Y 469.103,Z 472.529,A -85,B 0,C 180,E1 -7627.075,E2 -7627.075} C_VEL
LIN {X 0,Y 468.478,Z 487.015,A -85,B 0,C 180,E1 -7630.273,E2 -7630.273} C_VEL
LIN {X 0,Y 467.94,Z 499.207,A -85,B 0,C 180,E1 -7632.942,E2 -7632.942} C_VEL
LIN {X 0,Y 468.451,Z 502.366,A -85,B 0,C 180,E1 -7633.057,E2 -7633.057} C_VEL
LIN {X 0,Y 471.221,Z 519.183,A -85,B 0,C 180,E1 -7633.421,E2 -7633.421} C_VEL
LIN {X 0,Y 470.586,Z 604.178,A -85,B 0,C 180,E1 -7634.739,E2 -7634.739} C_VEL
LIN {X 0,Y 470.344,Z 614.096,A -85,B 0,C 180,E1 -7634.98,E2 -7634.98} C_VEL
LIN {X 0,Y 470.034,Z 624.086,A -85,B 0,C 180,E1 -7635.33,E2 -7635.33} C_VEL
LIN {X 0,Y 469.659,Z 634.446,A -85,B 0,C 180,E1 -7635.816,E2 -7635.816} C_VEL
LIN {X 0,Y 469.244,Z 643.913,A -85,B 0,C 180,E1 -7636.378,E2 -7636.378} C_VEL
LIN {X 0,Y 468.871,Z 652.6,A -85,B 0,C 180,E1 -7637.007,E2 -7637.007} C_VEL
LIN {X 0,Y 468.579,Z 660.498,A -85,B 0,C 180,E1 -7637.686,E2 -7637.686} C_VEL
LIN {X 0,Y 468.141,Z 668.756,A -85,B 0,C 180,E1 -7638.527,E2 -7638.527} C_VEL
LIN {X 0,Y 467.635,Z 677.553,A -85,B 0,C 180,E1 -7639.61,E2 -7639.61} C_VEL
LIN {X 0,Y 467.388,Z 683.545,A -85,B 0,C 180,E1 -7640.479,E2 -7640.479} C_VEL
LIN {X 0,Y 467.128,Z 689.857,A -85,B 0,C 180,E1 -7641.565,E2 -7641.565} C_VEL
LIN {X 0,Y 466.949,Z 695.131,A -85,B 0,C 180,E1 -7642.65,E2 -7642.65} C_VEL
LIN {X 0,Y 466.76,Z 700.222,A -85,B 0,C 180,E1 -7643.95,E2 -7643.95} C_VEL
LIN {X 0,Y 466.691,Z 704.183,A -85,B 0,C 180,E1 -7645.249,E2 -7645.249} C_VEL
LIN {X 0,Y 466.69,Z 707.114,A -85,B 0,C 180,E1 -7646.547,E2 -7646.547} C_VEL
LIN {X 0,Y 466.663,Z 708.611,A -85,B 0,C 180,E1 -7647.411,E2 -7647.411} C_VEL
LIN {X 0,Y 466.619,Z 710.129,A -85,B 0,C 180,E1 -7649.137,E2 -7649.137} C_VEL
LIN {X 0,Y 466.599,Z 710.407,A -85,B 0,C 180,E1 -7650,E2 -7650} C_VEL
LIN {X 0,Y 466.608,Z 709.535,A -85,B 0,C 180,E1 -7651.726,E2 -7651.726} C_VEL
LIN {X 0,Y 466.663,Z 708.611,A -85,B 0,C 180,E1 -7652.589,E2 -7652.589} C_VEL
LIN {X 0,Y 466.648,Z 705.27,A -85,B 0,C 180,E1 -7654.319,E2 -7654.319} C_VEL
LIN {X 0,Y 466.77,Z 701.65,A -85,B 0,C 180,E1 -7655.616,E2 -7655.616} C_VEL
LIN {X 0,Y 466.807,Z 698.841,A -85,B 0,C 180,E1 -7656.45,E2 -7656.45} C_VEL
LIN {X 0,Y 466.999,Z 693.134,A -85,B 0,C 180,E1 -7657.784,E2 -7657.784} C_VEL
LIN {X 0,Y 467.23,Z 687.482,A -85,B 0,C 180,E1 -7658.869,E2 -7658.869} C_VEL
LIN {X 0,Y 467.544,Z 680.677,A -85,B 0,C 180,E1 -7659.954,E2 -7659.954} C_VEL
LIN {X 0,Y 467.928,Z 672.457,A -85,B 0,C 180,E1 -7661.04,E2 -7661.04} C_VEL
LIN {X 0,Y 468.357,Z 664.629,A -85,B 0,C 180,E1 -7661.907,E2 -7661.907} C_VEL
LIN {X 0,Y 468.729,Z 656.558,A -85,B 0,C 180,E1 -7662.665,E2 -7662.665} C_VEL
LIN {X 0,Y 469.073,Z 648.531,A -85,B 0,C 180,E1 -7663.307,E2 -7663.307} C_VEL
LIN {X 0,Y 469.48,Z 638.383,A -85,B 0,C 180,E1 -7663.968,E2 -7663.968} C_VEL
LIN {X 0,Y 469.925,Z 627.875,A -85,B 0,C 180,E1 -7664.507,E2 -7664.507} C_VEL
LIN {X 0,Y 470.283,Z 617.542,A -85,B 0,C 180,E1 -7664.911,E2 -7664.911} C_VEL
LIN {X 0,Y 470.49,Z 606.82,A -85,B 0,C 180,E1 -7665.209,E2 -7665.209} C_VEL
LIN {X 0,Y 470.801,Z 585.838,A -85,B 0,C 180,E1 -7665.559,E2 -7665.559} C_VEL
LIN {X 0,Y 471.101,Z 517.733,A -85,B 0,C 180,E1 -7666.606,E2 -7666.606} C_VEL
LIN {X 0,Y 467.98,Z 499.607,A -85,B 0,C 180,E1 -7667.022,E2 -7667.022} C_VEL
LIN {X 0,Y 467.948,Z 498.087,A -85,B 0,C 180,E1 -7667.277,E2 -7667.277} C_VEL
LIN {X 0,Y 468.481,Z 487.156,A -85,B 0,C 180,E1 -7669.727,E2 -7669.727} C_VEL
LIN {X 0,Y 469.102,Z 472.59,A -85,B 0,C 180,E1 -7672.925,E2 -7672.925} C_VEL
LIN {X 0,Y 469.455,Z 463.236,A -85,B 0,C 180,E1 -7675.019,E2 -7675.019} C_VEL
LIN {X 0,Y 467.599,Z 452.865,A -85,B 0,C 180,E1 -7677.57,E2 -7677.57} C_VEL
LIN {X 0,Y 467.544,Z 452.746,A -85,B 0,C 180,E1 -7681.038,E2 -7681.038} C_VEL
LIN {X 0,Y 467.577,Z 452.745,A -85,B 0,C 180,E1 -7684.239,E2 -7684.239} C_VEL
LIN {X 0,Y 467.515,Z 452.744,A -85,B 0,C 180,E1 -7687.18,E2 -7687.18} C_VEL
LIN {X 0,Y 467.519,Z 452.738,A -85,B 0,C 180,E1 -7690.27,E2 -7690.27} C_VEL
LIN {X 0,Y 467.517,Z 452.747,A -85,B 0,C 180,E1 -7692.568,E2 -7692.568} C_VEL
LIN {X 0,Y 467.562,Z 452.738,A -85,B 0,C 180,E1 -7695.051,E2 -7695.051} C_VEL
LIN {X 0,Y 467.55,Z 452.741,A -85,B 0,C 180,E1 -7698.727,E2 -7698.727} C_VEL
LIN {X 0,Y 467.536,Z 452.746,A -85,B 0,C 180,E1 -7701.952,E2 -7701.952} C_VEL
LIN {X 0,Y 467.549,Z 452.736,A -85,B 0,C 180,E1 -7705.165,E2 -7705.165} C_VEL
LIN {X 0,Y 467.571,Z 452.744,A -85,B 0,C 180,E1 -7708.258,E2 -7708.258} C_VEL
LIN {X 0,Y 467.541,Z 452.74,A -85,B 0,C 180,E1 -7711.247,E2 -7711.247} C_VEL
LIN {X 0,Y 467.574,Z 452.737,A -85,B 0,C 180,E1 -7714.4,E2 -7714.4} C_VEL
LIN {X 0,Y 467.569,Z 452.738,A -85,B 0,C 180,E1 -7716.994,E2 -7716.994} C_VEL
LIN {X 0,Y 467.532,Z 452.743,A -85,B 0,C 180,E1 -7719.772,E2 -7719.772} C_VEL
LIN {X 0,Y 467.547,Z 452.736,A -85,B 0,C 180,E1 -7722.503,E2 -7722.503} C_VEL
LIN {X 0,Y 467.557,Z 452.738,A -85,B 0,C 180,E1 -7725.194,E2 -7725.194} C_VEL
LIN {X 0,Y 467.644,Z 452.732,A -85,B 0,C 180,E1 -7727.853,E2 -7727.853} C_VEL
LIN {X 0,Y 467.625,Z 452.716,A -85,B 0,C 180,E1 -7731.355,E2 -7731.355} C_VEL
LIN {X 0,Y 467.694,Z 452.725,A -85,B 0,C 180,E1 -7733.961,E2 -7733.961} C_VEL
LIN {X 0,Y 467.805,Z 452.708,A -85,B 0,C 180,E1 -7737.416,E2 -7737.416} C_VEL
LIN {X 0,Y 467.843,Z 452.694,A -85,B 0,C 180,E1 -7739.999,E2 -7739.999} C_VEL
LIN {X 0,Y 467.804,Z 452.707,A -85,B 0,C 180,E1 -7742.582,E2 -7742.582} C_VEL
LIN {X 0,Y 467.694,Z 452.73,A -85,B 0,C 180,E1 -7746.037,E2 -7746.037} C_VEL
LIN {X 0,Y 467.622,Z 452.722,A -85,B 0,C 180,E1 -7748.642,E2 -7748.642} C_VEL
LIN {X 0,Y 467.639,Z 452.728,A -85,B 0,C 180,E1 -7752.144,E2 -7752.144} C_VEL
LIN {X 0,Y 467.596,Z 452.739,A -85,B 0,C 180,E1 -7755.695,E2 -7755.695} C_VEL
LIN {X 0,Y 467.56,Z 452.726,A -85,B 0,C 180,E1 -7758.745,E2 -7758.745} C_VEL
LIN {X 0,Y 467.559,Z 452.735,A -85,B 0,C 180,E1 -7761.263,E2 -7761.263} C_VEL
LIN {X 0,Y 467.545,Z 452.748,A -85,B 0,C 180,E1 -7763.943,E2 -7763.943} C_VEL
LIN {X 0,Y 467.518,Z 452.735,A -85,B 0,C 180,E1 -7766.805,E2 -7766.805} C_VEL
LIN {X 0,Y 467.529,Z 452.744,A -85,B 0,C 180,E1 -7769.738,E2 -7769.738} C_VEL
LIN {X 0,Y 467.56,Z 452.738,A -85,B 0,C 180,E1 -7772.758,E2 -7772.758} C_VEL
LIN {X 0,Y 467.529,Z 452.742,A -85,B 0,C 180,E1 -7775.89,E2 -7775.89} C_VEL
LIN {X 0,Y 467.529,Z 452.743,A -85,B 0,C 180,E1 -7779.148,E2 -7779.148} C_VEL
LIN {X 0,Y 467.545,Z 452.736,A -85,B 0,C 180,E1 -7781.404,E2 -7781.404} C_VEL
LIN {X 0,Y 467.549,Z 452.738,A -85,B 0,C 180,E1 -7784.947,E2 -7784.947} C_VEL
LIN {X 0,Y 467.534,Z 452.728,A -85,B 0,C 180,E1 -7788.593,E2 -7788.593} C_VEL
LIN {X 0,Y 467.523,Z 452.751,A -85,B 0,C 180,E1 -7791.952,E2 -7791.952} C_VEL
LIN {X 0,Y 467.534,Z 452.73,A -85,B 0,C 180,E1 -7795.165,E2 -7795.165} C_VEL
LIN {X 0,Y 467.538,Z 452.748,A -85,B 0,C 180,E1 -7798.257,E2 -7798.257} C_VEL
LIN {X 0,Y 467.526,Z 452.737,A -85,B 0,C 180,E1 -7801.247,E2 -7801.247} C_VEL
LIN {X 0,Y 467.561,Z 452.745,A -85,B 0,C 180,E1 -7804.4,E2 -7804.4} C_VEL
LIN {X 0,Y 467.555,Z 452.742,A -85,B 0,C 180,E1 -7806.995,E2 -7806.995} C_VEL
LIN {X 0,Y 467.602,Z 452.742,A -85,B 0,C 180,E1 -7809.776,E2 -7809.776} C_VEL
LIN {X 0,Y 467.549,Z 452.746,A -85,B 0,C 180,E1 -7812.505,E2 -7812.505} C_VEL
LIN {X 0,Y 467.568,Z 452.742,A -85,B 0,C 180,E1 -7815.386,E2 -7815.386} C_VEL
LIN {X 0,Y 466.897,Z 452.829,A -85,B 0,C 180,E1 -7816.106,E2 -7816.106} C_VEL
LIN {X 0,Y 464.054,Z 453.18,A -85,B 0,C 180,E1 -7817.274,E2 -7817.274} C_VEL
LIN {X 0,Y 461.652,Z 453.483,A -85,B 0,C 180,E1 -7818.217,E2 -7818.217} C_VEL
LIN {X 0,Y 460.62,Z 453.608,A -85,B 0,C 180,E1 -7818.944,E2 -7818.944} C_VEL
LIN {X 0,Y 460.536,Z 453.619,A -85,B 0,C 180,E1 -7819.191,E2 -7819.191} C_VEL
LIN {X 0,Y 460.646,Z 453.607,A -85,B 0,C 180,E1 -7822.594,E2 -7822.594} C_VEL
LIN {X 0,Y 460.657,Z 453.604,A -85,B 0,C 180,E1 -7824.748,E2 -7824.748} C_VEL
LIN {X 0,Y 460.739,Z 453.594,A -85,B 0,C 180,E1 -7827.377,E2 -7827.377} C_VEL
LIN {X 0,Y 460.802,Z 453.589,A -85,B 0,C 180,E1 -7830,E2 -7830} C_VEL
LIN {X 0,Y 460.739,Z 453.594,A -85,B 0,C 180,E1 -7832.623,E2 -7832.623} C_VEL
LIN {X 0,Y 460.651,Z 453.608,A -85,B 0,C 180,E1 -7836.131,E2 -7836.131} C_VEL
LIN {X 0,Y 460.587,Z 453.612,A -85,B 0,C 180,E1 -7838.777,E2 -7838.777} C_VEL
LIN {X 0,Y 460.58,Z 453.615,A -85,B 0,C 180,E1 -7842.435,E2 -7842.435} C_VEL
LIN {X 0,Y 460.541,Z 453.621,A -85,B 0,C 180,E1 -7845.979,E2 -7845.979} C_VEL
LIN {X 0,Y 460.548,Z 453.619,A -85,B 0,C 180,E1 -7849.616,E2 -7849.616} C_VEL
LIN {X 0,Y 460.49,Z 453.625,A -85,B 0,C 180,E1 -7852.429,E2 -7852.429} C_VEL
LIN {X 0,Y 460.518,Z 453.624,A -85,B 0,C 180,E1 -7855.794,E2 -7855.794} C_VEL
LIN {X 0,Y 460.503,Z 453.611,A -85,B 0,C 180,E1 -7859.233,E2 -7859.233} C_VEL
LIN {X 0,Y 460.499,Z 453.622,A -85,B 0,C 180,E1 -7862.287,E2 -7862.287} C_VEL
LIN {X 0,Y 460.484,Z 453.61,A -85,B 0,C 180,E1 -7865.448,E2 -7865.448} C_VEL
LIN {X 0,Y 460.467,Z 453.623,A -85,B 0,C 180,E1 -7868.889,E2 -7868.889} C_VEL
LIN {X 0,Y 460.456,Z 453.606,A -85,B 0,C 180,E1 -7872.188,E2 -7872.188} C_VEL
LIN {X 0,Y 460.496,Z 453.618,A -85,B 0,C 180,E1 -7875.411,E2 -7875.411} C_VEL
LIN {X 0,Y 460.501,Z 453.612,A -85,B 0,C 180,E1 -7878.988,E2 -7878.988} C_VEL
LIN {X 0,Y 460.469,Z 453.626,A -85,B 0,C 180,E1 -7882.376,E2 -7882.376} C_VEL
LIN {X 0,Y 460.52,Z 453.611,A -85,B 0,C 180,E1 -7885.624,E2 -7885.624} C_VEL
LIN {X 0,Y 460.492,Z 453.621,A -85,B 0,C 180,E1 -7888.743,E2 -7888.743} C_VEL
LIN {X 0,Y 460.494,Z 453.616,A -85,B 0,C 180,E1 -7891.765,E2 -7891.765} C_VEL
LIN {X 0,Y 460.508,Z 453.617,A -85,B 0,C 180,E1 -7894.704,E2 -7894.704} C_VEL
LIN {X 0,Y 460.496,Z 453.623,A -85,B 0,C 180,E1 -7897.572,E2 -7897.572} C_VEL
LIN {X 0,Y 460.508,Z 453.605,A -85,B 0,C 180,E1 -7900.383,E2 -7900.383} C_VEL
LIN {X 0,Y 460.486,Z 453.617,A -85,B 0,C 180,E1 -7903.145,E2 -7903.145} C_VEL
LIN {X 0,Y 460.529,Z 453.623,A -85,B 0,C 180,E1 -7905.869,E2 -7905.869} C_VEL
LIN {X 0,Y 460.583,Z 453.598,A -85,B 0,C 180,E1 -7908.56,E2 -7908.56} C_VEL
LIN {X 0,Y 460.615,Z 453.605,A -85,B 0,C 180,E1 -7912.109,E2 -7912.109} C_VEL
LIN {X 0,Y 460.666,Z 453.598,A -85,B 0,C 180,E1 -7914.749,E2 -7914.749} C_VEL
LIN {X 0,Y 460.748,Z 453.585,A -85,B 0,C 180,E1 -7917.379,E2 -7917.379} C_VEL
LIN {X 0,Y 460.791,Z 453.572,A -85,B 0,C 180,E1 -7920.001,E2 -7920.001} C_VEL
LIN {X 0,Y 460.749,Z 453.587,A -85,B 0,C 180,E1 -7922.624,E2 -7922.624} C_VEL
LIN {X 0,Y 460.66,Z 453.599,A -85,B 0,C 180,E1 -7926.132,E2 -7926.132} C_VEL
LIN {X 0,Y 460.58,Z 453.593,A -85,B 0,C 180,E1 -7928.778,E2 -7928.778} C_VEL
LIN {X 0,Y 460.594,Z 453.607,A -85,B 0,C 180,E1 -7932.436,E2 -7932.436} C_VEL
LIN {X 0,Y 460.523,Z 453.615,A -85,B 0,C 180,E1 -7935.966,E2 -7935.966} C_VEL
LIN {X 0,Y 460.523,Z 453.602,A -85,B 0,C 180,E1 -7938.886,E2 -7938.886} C_VEL
LIN {X 0,Y 460.5,Z 453.62,A -85,B 0,C 180,E1 -7942.43,E2 -7942.43} C_VEL
LIN {X 0,Y 460.518,Z 453.613,A -85,B 0,C 180,E1 -7945.298,E2 -7945.298} C_VEL
LIN {X 0,Y 460.504,Z 453.62,A -85,B 0,C 180,E1 -7948.237,E2 -7948.237} C_VEL
LIN {X 0,Y 460.52,Z 453.618,A -85,B 0,C 180,E1 -7951.284,E2 -7951.284} C_VEL
LIN {X 0,Y 460.518,Z 453.613,A -85,B 0,C 180,E1 -7954.504,E2 -7954.504} C_VEL
LIN {X 0,Y 460.48,Z 453.626,A -85,B 0,C 180,E1 -7957.626,E2 -7957.626} C_VEL
LIN {X 0,Y 460.499,Z 453.618,A -85,B 0,C 180,E1 -7961.016,E2 -7961.016} C_VEL
LIN {X 0,Y 460.508,Z 453.618,A -85,B 0,C 180,E1 -7964.591,E2 -7964.591} C_VEL
LIN {X 0,Y 460.472,Z 453.621,A -85,B 0,C 180,E1 -7967.813,E2 -7967.813} C_VEL
LIN {X 0,Y 460.484,Z 453.621,A -85,B 0,C 180,E1 -7971.113,E2 -7971.113} C_VEL
LIN {X 0,Y 460.495,Z 453.621,A -85,B 0,C 180,E1 -7974.553,E2 -7974.553} C_VEL
LIN {X 0,Y 460.502,Z 453.62,A -85,B 0,C 180,E1 -7977.714,E2 -7977.714} C_VEL
LIN {X 0,Y 460.515,Z 453.623,A -85,B 0,C 180,E1 -7980.768,E2 -7980.768} C_VEL
LIN {X 0,Y 460.595,Z 453.853,A -85,B 0,C 180,E1 -7982.252,E2 -7982.252} C_VEL
LIN {X 0,Y 462.416,Z 464.115,A -85,B 0,C 180,E1 -7984.814,E2 -7984.814} C_VEL
LIN {X 0,Y 462.302,Z 470.281,A -85,B 0,C 180,E1 -7986.243,E2 -7986.243} C_VEL
LIN {X 0,Y 461.623,Z 483.74,A -85,B 0,C 180,E1 -7989.27,E2 -7989.27} C_VEL
LIN {X 0,Y 461.026,Z 497.029,A -85,B 0,C 180,E1 -7992.249,E2 -7992.249} C_VEL
LIN {X 0,Y 460.931,Z 499.018,A -85,B 0,C 180,E1 -7992.674,E2 -7992.674} C_VEL
LIN {X 0,Y 461.535,Z 502.535,A -85,B 0,C 180,E1 -7992.801,E2 -7992.801} C_VEL
LIN {X 0,Y 464.415,Z 519.393,A -85,B 0,C 180,E1 -7993.177,E2 -7993.177} C_VEL
LIN {X 0,Y 463.764,Z 603.982,A -85,B 0,C 180,E1 -7994.509,E2 -7994.509} C_VEL
LIN {X 0,Y 463.502,Z 613.901,A -85,B 0,C 180,E1 -7994.753,E2 -7994.753} C_VEL
LIN {X 0,Y 463.167,Z 623.89,A -85,B 0,C 180,E1 -7995.108,E2 -7995.108} C_VEL
LIN {X 0,Y 462.75,Z 634.249,A -85,B 0,C 180,E1 -7995.6,E2 -7995.6} C_VEL
LIN {X 0,Y 462.347,Z 643.398,A -85,B 0,C 180,E1 -7996.148,E2 -7996.148} C_VEL
LIN {X 0,Y 461.903,Z 652.943,A -85,B 0,C 180,E1 -7996.853,E2 -7996.853} C_VEL
LIN {X 0,Y 461.608,Z 660.499,A -85,B 0,C 180,E1 -7997.517,E2 -7997.517} C_VEL
LIN {X 0,Y 461.139,Z 668.559,A -85,B 0,C 180,E1 -7998.35,E2 -7998.35} C_VEL
LIN {X 0,Y 460.62,Z 677.356,A -85,B 0,C 180,E1 -7999.45,E2 -7999.45} C_VEL
LIN {X 0,Y 460.366,Z 683.349,A -85,B 0,C 180,E1 -8000.333,E2 -8000.333} C_VEL
LIN {X 0,Y 460.061,Z 689.66,A -85,B 0,C 180,E1 -8001.434,E2 -8001.434} C_VEL
LIN {X 0,Y 459.866,Z 694.934,A -85,B 0,C 180,E1 -8002.536,E2 -8002.536} C_VEL
LIN {X 0,Y 459.669,Z 700.025,A -85,B 0,C 180,E1 -8003.856,E2 -8003.856} C_VEL
LIN {X 0,Y 459.619,Z 703.987,A -85,B 0,C 180,E1 -8005.176,E2 -8005.176} C_VEL
LIN {X 0,Y 459.585,Z 706.918,A -85,B 0,C 180,E1 -8006.493,E2 -8006.493} C_VEL
LIN {X 0,Y 459.585,Z 708.415,A -85,B 0,C 180,E1 -8007.371,E2 -8007.371} C_VEL
LIN {X 0,Y 459.522,Z 709.933,A -85,B 0,C 180,E1 -8009.124,E2 -8009.124} C_VEL
LIN {X 0,Y 459.531,Z 710.212,A -85,B 0,C 180,E1 -8010,E2 -8010} C_VEL
LIN {X 0,Y 459.521,Z 709.339,A -85,B 0,C 180,E1 -8011.753,E2 -8011.753} C_VEL
LIN {X 0,Y 459.585,Z 708.415,A -85,B 0,C 180,E1 -8012.629,E2 -8012.629} C_VEL
LIN {X 0,Y 459.566,Z 705.074,A -85,B 0,C 180,E1 -8014.385,E2 -8014.385} C_VEL
LIN {X 0,Y 459.668,Z 701.452,A -85,B 0,C 180,E1 -8015.703,E2 -8015.703} C_VEL
LIN {X 0,Y 459.719,Z 698.513,A -85,B 0,C 180,E1 -8016.583,E2 -8016.583} C_VEL
LIN {X 0,Y 459.941,Z 692.938,A -85,B 0,C 180,E1 -8017.904,E2 -8017.904} C_VEL
LIN {X 0,Y 460.163,Z 687.284,A -85,B 0,C 180,E1 -8019.006,E2 -8019.006} C_VEL
LIN {X 0,Y 460.495,Z 680.479,A -85,B 0,C 180,E1 -8020.108,E2 -8020.108} C_VEL
LIN {X 0,Y 460.936,Z 672.26,A -85,B 0,C 180,E1 -8021.21,E2 -8021.21} C_VEL
LIN {X 0,Y 461.392,Z 664.432,A -85,B 0,C 180,E1 -8022.09,E2 -8022.09} C_VEL
LIN {X 0,Y 461.808,Z 655.412,A -85,B 0,C 180,E1 -8022.939,E2 -8022.939} C_VEL
LIN {X 0,Y 462.225,Z 646.58,A -85,B 0,C 180,E1 -8023.631,E2 -8023.631} C_VEL
LIN {X 0,Y 462.574,Z 638.186,A -85,B 0,C 180,E1 -8024.181,E2 -8024.181} C_VEL
LIN {X 0,Y 463.045,Z 627.679,A -85,B 0,C 180,E1 -8024.728,E2 -8024.728} C_VEL
LIN {X 0,Y 463.434,Z 617.346,A -85,B 0,C 180,E1 -8025.137,E2 -8025.137} C_VEL
LIN {X 0,Y 463.64,Z 606.624,A -85,B 0,C 180,E1 -8025.439,E2 -8025.439} C_VEL
LIN {X 0,Y 463.974,Z 585.642,A -85,B 0,C 180,E1 -8025.794,E2 -8025.794} C_VEL
LIN {X 0,Y 464.305,Z 518.595,A -85,B 0,C 180,E1 -8026.84,E2 -8026.84} C_VEL
LIN {X 0,Y 460.954,Z 499.475,A -85,B 0,C 180,E1 -8027.286,E2 -8027.286} C_VEL
LIN {X 0,Y 460.95,Z 498.321,A -85,B 0,C 180,E1 -8027.445,E2 -8027.445} C_VEL
LIN {X 0,Y 461.47,Z 486.989,A -85,B 0,C 180,E1 -8030.039,E2 -8030.039} C_VEL
LIN {X 0,Y 462.064,Z 474.546,A -85,B 0,C 180,E1 -8032.821,E2 -8032.821} C_VEL
LIN {X 0,Y 462.525,Z 465.14,A -85,B 0,C 180,E1 -8034.939,E2 -8034.939} C_VEL
LIN {X 0,Y 461.153,Z 456.93,A -85,B 0,C 180,E1 -8036.961,E2 -8036.961} C_VEL
LIN {X 0,Y 460.574,Z 453.734,A -85,B 0,C 180,E1 -8037.798,E2 -8037.798} C_VEL
LIN {X 0,Y 460.523,Z 453.621,A -85,B 0,C 180,E1 -8041.282,E2 -8041.282} C_VEL
LIN {X 0,Y 460.521,Z 453.62,A -85,B 0,C 180,E1 -8044.502,E2 -8044.502} C_VEL
LIN {X 0,Y 460.483,Z 453.622,A -85,B 0,C 180,E1 -8047.624,E2 -8047.624} C_VEL
LIN {X 0,Y 460.5,Z 453.607,A -85,B 0,C 180,E1 -8051.014,E2 -8051.014} C_VEL
LIN {X 0,Y 460.507,Z 453.619,A -85,B 0,C 180,E1 -8054.589,E2 -8054.589} C_VEL
LIN {X 0,Y 460.471,Z 453.627,A -85,B 0,C 180,E1 -8057.812,E2 -8057.812} C_VEL
LIN {X 0,Y 460.481,Z 453.618,A -85,B 0,C 180,E1 -8061.111,E2 -8061.111} C_VEL
LIN {X 0,Y 460.499,Z 453.617,A -85,B 0,C 180,E1 -8064.552,E2 -8064.552} C_VEL
LIN {X 0,Y 460.521,Z 453.614,A -85,B 0,C 180,E1 -8067.714,E2 -8067.714} C_VEL
LIN {X 0,Y 460.518,Z 453.616,A -85,B 0,C 180,E1 -8070.766,E2 -8070.766} C_VEL
LIN {X 0,Y 460.531,Z 453.61,A -85,B 0,C 180,E1 -8074.207,E2 -8074.207} C_VEL
LIN {X 0,Y 460.541,Z 453.615,A -85,B 0,C 180,E1 -8076.623,E2 -8076.623} C_VEL
LIN {X 0,Y 460.478,Z 453.619,A -85,B 0,C 180,E1 -8079.448,E2 -8079.448} C_VEL
LIN {X 0,Y 460.503,Z 453.61,A -85,B 0,C 180,E1 -8082.227,E2 -8082.227} C_VEL
LIN {X 0,Y 460.515,Z 453.615,A -85,B 0,C 180,E1 -8084.962,E2 -8084.962} C_VEL
LIN {X 0,Y 460.6,Z 453.607,A -85,B 0,C 180,E1 -8087.664,E2 -8087.664} C_VEL
LIN {X 0,Y 460.58,Z 453.593,A -85,B 0,C 180,E1 -8091.222,E2 -8091.222} C_VEL
LIN {X 0,Y 460.66,Z 453.599,A -85,B 0,C 180,E1 -8093.868,E2 -8093.868} C_VEL
LIN {X 0,Y 460.749,Z 453.587,A -85,B 0,C 180,E1 -8097.376,E2 -8097.376} C_VEL
LIN {X 0,Y 460.791,Z 453.572,A -85,B 0,C 180,E1 -8099.999,E2 -8099.999} C_VEL
LIN {X 0,Y 460.748,Z 453.585,A -85,B 0,C 180,E1 -8102.621,E2 -8102.621} C_VEL
LIN {X 0,Y 460.66,Z 453.604,A -85,B 0,C 180,E1 -8106.129,E2 -8106.129} C_VEL
LIN {X 0,Y 460.577,Z 453.599,A -85,B 0,C 180,E1 -8108.776,E2 -8108.776} C_VEL
LIN {X 0,Y 460.589,Z 453.609,A -85,B 0,C 180,E1 -8112.434,E2 -8112.434} C_VEL
LIN {X 0,Y 460.549,Z 453.619,A -85,B 0,C 180,E1 -8115.977,E2 -8115.977} C_VEL
LIN {X 0,Y 460.519,Z 453.602,A -85,B 0,C 180,E1 -8118.884,E2 -8118.884} C_VEL
LIN {X 0,Y 460.503,Z 453.615,A -85,B 0,C 180,E1 -8121.484,E2 -8121.484} C_VEL
LIN {X 0,Y 460.505,Z 453.621,A -85,B 0,C 180,E1 -8124.333,E2 -8124.333} C_VEL
LIN {X 0,Y 460.476,Z 453.611,A -85,B 0,C 180,E1 -8127.248,E2 -8127.248} C_VEL
LIN {X 0,Y 460.489,Z 453.627,A -85,B 0,C 180,E1 -8130.24,E2 -8130.24} C_VEL
LIN {X 0,Y 460.503,Z 453.617,A -85,B 0,C 180,E1 -8133.325,E2 -8133.325} C_VEL
LIN {X 0,Y 460.446,Z 453.628,A -85,B 0,C 180,E1 -8136.53,E2 -8136.53} C_VEL
LIN {X 0,Y 460.496,Z 453.621,A -85,B 0,C 180,E1 -8139.864,E2 -8139.864} C_VEL
LIN {X 0,Y 460.447,Z 453.626,A -85,B 0,C 180,E1 -8142.892,E2 -8142.892} C_VEL
LIN {X 0,Y 460.49,Z 453.617,A -85,B 0,C 180,E1 -8145.83,E2 -8145.83} C_VEL
LIN {X 0,Y 460.484,Z 453.607,A -85,B 0,C 180,E1 -8148.984,E2 -8148.984} C_VEL
LIN {X 0,Y 460.466,Z 453.627,A -85,B 0,C 180,E1 -8152.374,E2 -8152.374} C_VEL
LIN {X 0,Y 460.517,Z 453.605,A -85,B 0,C 180,E1 -8155.622,E2 -8155.622} C_VEL
LIN {X 0,Y 460.488,Z 453.622,A -85,B 0,C 180,E1 -8158.741,E2 -8158.741} C_VEL
LIN {X 0,Y 460.49,Z 453.618,A -85,B 0,C 180,E1 -8161.763,E2 -8161.763} C_VEL
LIN {X 0,Y 460.505,Z 453.622,A -85,B 0,C 180,E1 -8164.703,E2 -8164.703} C_VEL
LIN {X 0,Y 460.49,Z 453.625,A -85,B 0,C 180,E1 -8167.571,E2 -8167.571} C_VEL
LIN {X 0,Y 460.548,Z 453.619,A -85,B 0,C 180,E1 -8170.384,E2 -8170.384} C_VEL
LIN {X 0,Y 460.55,Z 453.62,A -85,B 0,C 180,E1 -8174.057,E2 -8174.057} C_VEL
LIN {X 0,Y 460.586,Z 453.615,A -85,B 0,C 180,E1 -8177.665,E2 -8177.665} C_VEL
LIN {X 0,Y 460.536,Z 453.619,A -85,B 0,C 180,E1 -8179.191,E2 -8179.191} C_VEL
LIN {X 0,Y 459.871,Z 453.705,A -85,B 0,C 180,E1 -8179.921,E2 -8179.921} C_VEL
LIN {X 0,Y 457.04,Z 454.058,A -85,B 0,C 180,E1 -8181.107,E2 -8181.107} C_VEL
LIN {X 0,Y 454.655,Z 454.355,A -85,B 0,C 180,E1 -8182.064,E2 -8182.064} C_VEL
LIN {X 0,Y 453.644,Z 454.478,A -85,B 0,C 180,E1 -8182.802,E2 -8182.802} C_VEL
LIN {X 0,Y 453.568,Z 454.487,A -85,B 0,C 180,E1 -8183.052,E2 -8183.052} C_VEL
LIN {X 0,Y 453.63,Z 454.48,A -85,B 0,C 180,E1 -8184.666,E2 -8184.666} C_VEL
LIN {X 0,Y 453.669,Z 454.477,A -85,B 0,C 180,E1 -8188.225,E2 -8188.225} C_VEL
LIN {X 0,Y 453.75,Z 454.467,A -85,B 0,C 180,E1 -8190,E2 -8190} C_VEL
LIN {X 0,Y 453.686,Z 454.473,A -85,B 0,C 180,E1 -8192.664,E2 -8192.664} C_VEL
LIN {X 0,Y 453.619,Z 454.484,A -85,B 0,C 180,E1 -8196.226,E2 -8196.226} C_VEL
LIN {X 0,Y 453.553,Z 454.488,A -85,B 0,C 180,E1 -8198.914,E2 -8198.914} C_VEL
LIN {X 0,Y 453.548,Z 454.49,A -85,B 0,C 180,E1 -8202.529,E2 -8202.529} C_VEL
LIN {X 0,Y 453.486,Z 454.5,A -85,B 0,C 180,E1 -8206.091,E2 -8206.091} C_VEL
LIN {X 0,Y 453.501,Z 454.494,A -85,B 0,C 180,E1 -8209.04,E2 -8209.04} C_VEL
LIN {X 0,Y 453.459,Z 454.503,A -85,B 0,C 180,E1 -8211.837,E2 -8211.837} C_VEL
LIN {X 0,Y 453.453,Z 454.5,A -85,B 0,C 180,E1 -8214.738,E2 -8214.738} C_VEL
LIN {X 0,Y 453.445,Z 454.5,A -85,B 0,C 180,E1 -8217.943,E2 -8217.943} C_VEL
LIN {X 0,Y 453.44,Z 454.499,A -85,B 0,C 180,E1 -8220.762,E2 -8220.762} C_VEL
LIN {X 0,Y 453.449,Z 454.488,A -85,B 0,C 180,E1 -8223.915,E2 -8223.915} C_VEL
LIN {X 0,Y 453.419,Z 454.501,A -85,B 0,C 180,E1 -8227.192,E2 -8227.192} C_VEL
LIN {X 0,Y 453.449,Z 454.484,A -85,B 0,C 180,E1 -8230.613,E2 -8230.613} C_VEL
LIN {X 0,Y 453.467,Z 454.494,A -85,B 0,C 180,E1 -8234.529,E2 -8234.529} C_VEL
LIN {X 0,Y 453.422,Z 454.501,A -85,B 0,C 180,E1 -8238.072,E2 -8238.072} C_VEL
LIN {X 0,Y 453.425,Z 454.5,A -85,B 0,C 180,E1 -8240.803,E2 -8240.803} C_VEL
LIN {X 0,Y 453.428,Z 454.501,A -85,B 0,C 180,E1 -8243.917,E2 -8243.917} C_VEL
LIN {X 0,Y 453.46,Z 454.494,A -85,B 0,C 180,E1 -8247.151,E2 -8247.151} C_VEL
LIN {X 0,Y 453.449,Z 454.497,A -85,B 0,C 180,E1 -8250.268,E2 -8250.268} C_VEL
LIN {X 0,Y 453.427,Z 454.49,A -85,B 0,C 180,E1 -8253.291,E2 -8253.291} C_VEL
LIN {X 0,Y 453.482,Z 454.498,A -85,B 0,C 180,E1 -8256.239,E2 -8256.239} C_VEL
LIN {X 0,Y 453.455,Z 454.491,A -85,B 0,C 180,E1 -8259.118,E2 -8259.118} C_VEL
LIN {X 0,Y 453.447,Z 454.49,A -85,B 0,C 180,E1 -8261.944,E2 -8261.944} C_VEL
LIN {X 0,Y 453.506,Z 454.491,A -85,B 0,C 180,E1 -8264.727,E2 -8264.727} C_VEL
LIN {X 0,Y 453.557,Z 454.484,A -85,B 0,C 180,E1 -8267.473,E2 -8267.473} C_VEL
LIN {X 0,Y 453.547,Z 454.473,A -85,B 0,C 180,E1 -8271.087,E2 -8271.087} C_VEL
LIN {X 0,Y 453.628,Z 454.479,A -85,B 0,C 180,E1 -8273.775,E2 -8273.775} C_VEL
LIN {X 0,Y 453.695,Z 454.464,A -85,B 0,C 180,E1 -8277.338,E2 -8277.338} C_VEL
LIN {X 0,Y 453.742,Z 454.449,A -85,B 0,C 180,E1 -8280.001,E2 -8280.001} C_VEL
LIN {X 0,Y 453.696,Z 454.465,A -85,B 0,C 180,E1 -8282.665,E2 -8282.665} C_VEL
LIN {X 0,Y 453.629,Z 454.474,A -85,B 0,C 180,E1 -8286.227,E2 -8286.227} C_VEL
LIN {X 0,Y 453.551,Z 454.467,A -85,B 0,C 180,E1 -8288.915,E2 -8288.915} C_VEL
LIN {X 0,Y 453.562,Z 454.482,A -85,B 0,C 180,E1 -8292.53,E2 -8292.53} C_VEL
LIN {X 0,Y 453.482,Z 454.489,A -85,B 0,C 180,E1 -8296.199,E2 -8296.199} C_VEL
LIN {X 0,Y 453.483,Z 454.478,A -85,B 0,C 180,E1 -8299.029,E2 -8299.029} C_VEL
LIN {X 0,Y 453.469,Z 454.498,A -85,B 0,C 180,E1 -8301.838,E2 -8301.838} C_VEL
LIN {X 0,Y 453.466,Z 454.49,A -85,B 0,C 180,E1 -8304.738,E2 -8304.738} C_VEL
LIN {X 0,Y 453.46,Z 454.492,A -85,B 0,C 180,E1 -8307.943,E2 -8307.943} C_VEL
LIN {X 0,Y 453.456,Z 454.497,A -85,B 0,C 180,E1 -8310.762,E2 -8310.762} C_VEL
LIN {X 0,Y 453.464,Z 454.491,A -85,B 0,C 180,E1 -8313.915,E2 -8313.915} C_VEL
LIN {X 0,Y 453.433,Z 454.5,A -85,B 0,C 180,E1 -8317.193,E2 -8317.193} C_VEL
LIN {X 0,Y 453.464,Z 454.495,A -85,B 0,C 180,E1 -8320.613,E2 -8320.613} C_VEL
LIN {X 0,Y 453.479,Z 454.494,A -85,B 0,C 180,E1 -8324.529,E2 -8324.529} C_VEL
LIN {X 0,Y 453.431,Z 454.493,A -85,B 0,C 180,E1 -8328.073,E2 -8328.073} C_VEL
LIN {X 0,Y 453.426,Z 454.5,A -85,B 0,C 180,E1 -8330.805,E2 -8330.805} C_VEL
LIN {X 0,Y 453.44,Z 454.496,A -85,B 0,C 180,E1 -8333.916,E2 -8333.916} C_VEL
LIN {X 0,Y 453.467,Z 454.493,A -85,B 0,C 180,E1 -8336.817,E2 -8336.817} C_VEL
LIN {X 0,Y 453.456,Z 454.5,A -85,B 0,C 180,E1 -8340.267,E2 -8340.267} C_VEL
LIN {X 0,Y 453.544,Z 454.67,A -85,B 0,C 180,E1 -8342.007,E2 -8342.007} C_VEL
LIN {X 0,Y 455.4,Z 464.995,A -85,B 0,C 180,E1 -8344.644,E2 -8344.644} C_VEL
LIN {X 0,Y 455.482,Z 468.786,A -85,B 0,C 180,E1 -8345.557,E2 -8345.557} C_VEL
LIN {X 0,Y 454.676,Z 483.566,A -85,B 0,C 180,E1 -8348.938,E2 -8348.938} C_VEL
LIN {X 0,Y 454.158,Z 494.886,A -85,B 0,C 180,E1 -8351.505,E2 -8351.505} C_VEL
LIN {X 0,Y 453.954,Z 498.823,A -85,B 0,C 180,E1 -8352.399,E2 -8352.399} C_VEL
LIN {X 0,Y 454.471,Z 502.004,A -85,B 0,C 180,E1 -8352.52,E2 -8352.52} C_VEL
LIN {X 0,Y 457.606,Z 520.45,A -85,B 0,C 180,E1 -8352.939,E2 -8352.939} C_VEL
LIN {X 0,Y 456.934,Z 603.786,A -85,B 0,C 180,E1 -8354.271,E2 -8354.271} C_VEL
LIN {X 0,Y 456.657,Z 613.704,A -85,B 0,C 180,E1 -8354.519,E2 -8354.519} C_VEL
LIN {X 0,Y 456.319,Z 623.694,A -85,B 0,C 180,E1 -8354.879,E2 -8354.879} C_VEL
LIN {X 0,Y 455.88,Z 634.053,A -85,B 0,C 180,E1 -8355.378,E2 -8355.378} C_VEL
LIN {X 0,Y 455.421,Z 643.201,A -85,B 0,C 180,E1 -8355.933,E2 -8355.933} C_VEL
LIN {X 0,Y 455.017,Z 652.207,A -85,B 0,C 180,E1 -8356.604,E2 -8356.604} C_VEL
LIN {X 0,Y 454.625,Z 660.488,A -85,B 0,C 180,E1 -8357.341,E2 -8357.341} C_VEL
LIN {X 0,Y 454.167,Z 668.362,A -85,B 0,C 180,E1 -8358.168,E2 -8358.168} C_VEL
LIN {X 0,Y 453.615,Z 677.159,A -85,B 0,C 180,E1 -8359.285,E2 -8359.285} C_VEL
LIN {X 0,Y 453.334,Z 683.151,A -85,B 0,C 180,E1 -8360.181,E2 -8360.181} C_VEL
LIN {X 0,Y 453.019,Z 689.463,A -85,B 0,C 180,E1 -8361.3,E2 -8361.3} C_VEL
LIN {X 0,Y 452.814,Z 694.737,A -85,B 0,C 180,E1 -8362.419,E2 -8362.419} C_VEL
LIN {X 0,Y 452.607,Z 699.828,A -85,B 0,C 180,E1 -8363.76,E2 -8363.76} C_VEL
LIN {X 0,Y 452.547,Z 703.791,A -85,B 0,C 180,E1 -8365.1,E2 -8365.1} C_VEL
LIN {X 0,Y 452.481,Z 706.721,A -85,B 0,C 180,E1 -8366.438,E2 -8366.438} C_VEL
LIN {X 0,Y 452.509,Z 708.22,A -85,B 0,C 180,E1 -8367.329,E2 -8367.329} C_VEL
LIN {X 0,Y 452.429,Z 709.737,A -85,B 0,C 180,E1 -8369.11,E2 -8369.11} C_VEL
LIN {X 0,Y 452.435,Z 710.016,A -85,B 0,C 180,E1 -8370,E2 -8370} C_VEL
LIN {X 0,Y 452.437,Z 709.143,A -85,B 0,C 180,E1 -8371.78,E2 -8371.78} C_VEL
LIN {X 0,Y 452.509,Z 708.22,A -85,B 0,C 180,E1 -8372.671,E2 -8372.671} C_VEL
LIN {X 0,Y 452.488,Z 704.877,A -85,B 0,C 180,E1 -8374.454,E2 -8374.454} C_VEL
LIN {X 0,Y 452.569,Z 702.667,A -85,B 0,C 180,E1 -8375.346,E2 -8375.346} C_VEL
LIN {X 0,Y 452.644,Z 698.488,A -85,B 0,C 180,E1 -8376.642,E2 -8376.642} C_VEL
LIN {X 0,Y 452.887,Z 692.741,A -85,B 0,C 180,E1 -8378.028,E2 -8378.028} C_VEL
LIN {X 0,Y 453.118,Z 687.087,A -85,B 0,C 180,E1 -8379.148,E2 -8379.148} C_VEL
LIN {X 0,Y 453.459,Z 680.281,A -85,B 0,C 180,E1 -8380.267,E2 -8380.267} C_VEL
LIN {X 0,Y 453.95,Z 672.064,A -85,B 0,C 180,E1 -8381.384,E2 -8381.384} C_VEL
LIN {X 0,Y 454.427,Z 664.235,A -85,B 0,C 180,E1 -8382.278,E2 -8382.278} C_VEL
LIN {X 0,Y 454.875,Z 655.215,A -85,B 0,C 180,E1 -8383.14,E2 -8383.14} C_VEL
LIN {X 0,Y 455.308,Z 646.383,A -85,B 0,C 180,E1 -8383.842,E2 -8383.842} C_VEL
LIN {X 0,Y 455.683,Z 637.99,A -85,B 0,C 180,E1 -8384.4,E2 -8384.4} C_VEL
